// TwinCAT 3 PLC project IDPLC
// ProgramVersion: 3.1.4024.12
// libraries:
//   Recipe Management, * (System)
//   Tc2_Drive, * (Beckhoff Automation GmbH)
//   Tc2_EtherCAT, * (Beckhoff Automation GmbH)
//   Tc2_Math, * (Beckhoff Automation GmbH)
//   Tc2_MC2, * (Beckhoff Automation GmbH)
//   Tc2_NC, * (Beckhoff Automation GmbH)
//   Tc2_NcDrive, * (Beckhoff Automation GmbH)
//   Tc2_SerialCom, * (Beckhoff Automation GmbH)
//   Tc2_Standard, * (Beckhoff Automation GmbH)
//   Tc2_System, * (Beckhoff Automation GmbH)
//   Tc2_Utilities, * (Beckhoff Automation GmbH)
//   Tc3_Module, * (Beckhoff Automation GmbH)
// project tree:
//   DUTs/ DUT.TcDUT (not stored), DUT_SENSOR_DATAS_1.TcDUT (not stored), DUT_SENSOR_DATAS_8.TcDUT (not stored), DUT_SENSOR_DATAS_2.TcDUT (not stored), DUT_SENSOR_DATAS_3.TcDUT (not stored), DUT_SENSOR_DATAS_4.TcDUT (not stored), DUT_SENSOR_DATAS_5.TcDUT (not stored), DUT_SENSOR_DATAS_6.TcDUT (not stored), DUT_SENSOR_DATAS_7.TcDUT (not stored), Struct_M_Compensation.TcDUT, Struct_M_lakeshore.TcDUT (not stored), ST_P180.TcDUT (not stored), ST_P182.TcDUT (not stored), ST_P183.TcDUT (not stored)
//   GVLs/ Global_Variables.TcGVL, Variable_Configuration.TcGVL (not stored)
//   / PlcTask.TcTTO (not stored), RecipeManager.TcRMO (not stored)
//   POUs/0.UserMode/ F_GetSysTime.TcPOU (not stored), UserMode.TcPOU
//   POUs/1.CarrierMode/SingleCarrierMode/ SingleCarrierMode.TcPOU
//   POUs/2.SingleMotorMode/DebugMode/ DebugMode.TcPOU
//   POUs/CommonFB/ExternFB/ FB_LedShow.TcPOU (not stored), FB_PlcEmergencyStop.TcPOU (not stored)
//   POUs/CommonFB/MainFB/ FB_Move.TcPOU, FB_Power.TcPOU, FB_SetAxisPosition.TcPOU, FB_SetMotorAxisPosition.TcPOU, FB_Stop.TcPOU
//   POUs/ MAIN.TcPOU
//   POUs/RS232/ BackgroundEL.TcPOU (not stored), FB_SerialCom.TcPOU (not stored)

// ---- DUTs/Struct_M_Compensation.TcDUT
TYPE Struct_M_Compensation :
STRUCT
	Encoder:LREAL;
	LeftTop:LREAL;
	RightTop:LREAL;
	LeftBottom:LREAL;
	RightBottom:LREAL;
	LeftIn:LREAL;
	RightIn:LREAL;
	LeftOut:LREAL;
	RightOut:LREAL;
	InRange:BOOL;
END_STRUCT
END_TYPE

// ---- GVLs/Global_Variables.TcGVL
//{attribute 'Tc2GvlVarNames'}
VAR_GLOBAL
(*IDControl Ready*)
	IDControlReady:BOOL;
(*RecipeDescription*)
	RecipeSavedDate:STRING;
	RecipeDescription:STRING;
(*key Command*)
	btn_Power:BOOL;
	btn_PowerOn: BOOL;
	btn_PowerOff: BOOL;
(*Reset*)
	btn_Reset:BOOL;
(*Error Massage*)
	Error:BOOL;
	ErrorID:DINT;
	ErrorDescription:STRING;
(*加载配方参数*)
	LoadRecipeParameters:BOOL;
	loadParametersDone:BOOL;
(*Max Velocity Global*)
	MaxVelocityGlobalVelocity : LREAL;
(*设置光栅bias done *)	
	PositionBiasDone:BOOL;
(*回程差*)
	HysteresisError:LREAL;
(*Drive Status*)
	DriveStatus:DINT;//1:Drive Ready;2:Axis is in operation;0:Others
(*光栅漂移误差阈值*)
	LEDriftErrorThreshold:LREAL:=0.001;
(*Lag Distance threshold*)
	PosDiff_LeftTopLin: LREAL:=0.5;
	PosDiff_RightTopLin:LREAL:=0.5;
	PosDiff_LeftBottomLin:LREAL:=0.5;
	PosDiff_RightBottomLin:LREAL:=0.5;	
	PosDiff_LeftInLin: LREAL:=0.5;
	PosDiff_RightInLin:LREAL:=0.5;
	PosDiff_LeftOutLin:LREAL:=0.5;
	PosDiff_RightOutLin:LREAL:=0.5;
(*UserMode Threshold*)
	Threshold_UserTopPos: LREAL:=0.5;
	Threshold_UserBottomPos: LREAL:=0.5;
	Threshold_UserTBLeftPos: LREAL:=0.5;//TB=Top&Bottom
	Threshold_UserTBRightPos: LREAL:=0.5;
	Threshold_UserTopVelo: LREAL:=0.5;
	Threshold_UserBottomVelo: LREAL:=0.5;
	Threshold_UserTBLeftVelo: LREAL:=0.5;
	Threshold_UserTBRightVelo: LREAL:=0.5;
	Threshold_UserInPos: LREAL:=0.5;
	Threshold_UserOutPos: LREAL:=0.5;
	Threshold_UserIOLeftPos: LREAL:=0.5;//IO=In&Out
	Threshold_UserIORightPos: LREAL:=0.5;
	Threshold_UserInVelo: LREAL:=0.5;
	Threshold_UserOutVelo: LREAL:=0.5;
	Threshold_UserIOLeftVelo: LREAL:=0.5;
	Threshold_UserIORightVelo: LREAL:=0.5;
	//
	Range_UserTBTaperPos:LREAL:=4.01;
	Range_UserTBTaperVelo:LREAL:=1.01;
	Range_UserIOTaperPos:LREAL:=4.01;
	Range_UserIOTaperVelo:LREAL:=1.01;
(*UserMode*)
	//UserGapPositionNew:LREAL:=20;//target
	//UserGapVelocityNew:LREAL:=1;//target
(*DebugMode Threshold*)
	Threshold_TopPos_Debug: LREAL:=4;
	Threshold_BottomPos_Debug: LREAL:=4;
	Threshold_TBLeftPos_Debug: LREAL:=4;
	Threshold_TBRightPos_Debug: LREAL:=4;
	Threshold_InPos_Debug: LREAL:=4;
	Threshold_OutPos_Debug: LREAL:=4;
	Threshold_IOLeftPos_Debug: LREAL:=4;
	Threshold_IORightPos_Debug: LREAL:=4;
(*SingleCarrierMode threshold*)
	Threshold_TopPos_SingleCarrier: LREAL:=2;
	Threshold_BottomPos_SingleCarrier: LREAL:=2;
	Threshold_TBLeftPos_SingleCarrier: LREAL:=2;
	Threshold_TBRightPos_SingleCarrier: LREAL:=2;
	Threshold_TopVelo_SingleCarrier: LREAL:=2;
	Threshold_BottomVelo_SingleCarrier: LREAL:=2;
	Threshold_TBLeftVelo_SingleCarrier: LREAL:=2;
	Threshold_TBRightVelo_SingleCarrier: LREAL:=2;
	Threshold_InPos_SingleCarrier: LREAL:=2;
	Threshold_OutPos_SingleCarrier: LREAL:=2;
	Threshold_IOLeftPos_SingleCarrier: LREAL:=2;
	Threshold_IORightPos_SingleCarrier: LREAL:=2;
	Threshold_InVelo_SingleCarrier: LREAL:=2;
	Threshold_OutVelo_SingleCarrier: LREAL:=2;
	Threshold_IOLeftVelo_SingleCarrier: LREAL:=2;
	Threshold_IORightVelo_SingleCarrier: LREAL:=2;
	
	moveDoneLeftTop: BOOL;
	moveDoneRightTop: BOOL;
	moveDoneLeftBottom: BOOL;
	moveDoneRightBottom: BOOL;
	moveDoneLeftIn: BOOL;
	moveDoneRightIn: BOOL;
	moveDoneLeftOut: BOOL;
	moveDoneRightOut: BOOL;
	moveDoneAllAxis: BOOL;
	moveStatusLeftTop: BOOL;
	moveStatusRightTop: BOOL;
	moveStatusLeftBottom: BOOL;
	moveStatusRightBottom: BOOL;
	moveStatusLeftIn: BOOL;
	moveStatusRightIn: BOOL;
	moveStatusLeftOut: BOOL;
	moveStatusRightOut: BOOL;
	moveStatusAllAxis: BOOL;
	moveStatusAnyAxis: BOOL;
	
	moveDoneLeftTopMotor: BOOL;
	moveDoneRightTopMotor: BOOL;
	moveDoneLeftBottomMotor: BOOL;
	moveDoneRightBottomMotor: BOOL;
	moveDoneLeftInMotor: BOOL;
	moveDoneRightInMotor: BOOL;
	moveDoneLeftOutMotor: BOOL;
	moveDoneRightOutMotor: BOOL;
	moveDoneAllAxisMotor: BOOL;
	moveStatusLeftTopMotor: BOOL;
	moveStatusRightTopMotor: BOOL;
	moveStatusLeftBottomMotor: BOOL;
	moveStatusRightBottomMotor: BOOL;
	moveStatusLeftInMotor: BOOL;
	moveStatusRightInMotor: BOOL;
	moveStatusLeftOutMotor: BOOL;
	moveStatusRightOutMotor: BOOL;
	moveStatusAllAxisMotor: BOOL;
	moveStatusAnyAxisMotor: BOOL;
	(*input protection*)
	//
	min_UserGapPositionNew:LREAL:=10;
	max_UserGapPositionNew:LREAL:=200;
	inRange_UserGapPositionNew:BOOL;
	//LE protection position
	min_UserLEProtectionGapPosition:LREAL;
	min_ThresholdGapSoft2LEProtection:LREAL;
	max_UserLEProtectionGapPosition:LREAL;
	max_ThresholdGapSoft2LEProtection:LREAL;
	//
	min_UserGapVelocityNew:LREAL:=0;
	max_UserGapVelocityNew:LREAL:=2;
	inRange_UserGapVelocityNew:BOOL;
	//
	min_UserTaperPositionNew: LREAL:=0;;
	max_UserTaperPositionNew: LREAL:=1;
	inRange_UserTaperPositionNew: BOOL;
	//
	min_UserTaperVelocityNew: LREAL:=0;
	max_UserTaperVelocityNew: LREAL:=1;
	inRange_UserTaperVelocityNew: BOOL;
	
(*Compensation Value*)
	M_Compensation:ARRAY[1..18] OF Struct_M_Compensation
:=[
(Encoder:=0,		LeftTop:=0,			RightTop:=0,		LeftBottom:=0,			RightBottom:=0,			
					LeftIn:=0,			RightIn:=0,			LeftOut:=0,				RightOut:=0,			InRange:=FALSE),
(Encoder:=5,		LeftTop:=5,			RightTop:=5,		LeftBottom:=5,			RightBottom:=5,			
					LeftIn:=5,			RightIn:=5,			LeftOut:=5,				RightOut:=5,			InRange:=FALSE),
(Encoder:=6,		LeftTop:=6,			RightTop:=6,		LeftBottom:=6,			RightBottom:=6,			
					LeftIn:=6,			RightIn:=6,			LeftOut:=6,				RightOut:=6,			InRange:=FALSE),
(Encoder:=7,		LeftTop:=7,			RightTop:=7,		LeftBottom:=7,			RightBottom:=7,			
					LeftIn:=7,			RightIn:=7,			LeftOut:=7,				RightOut:=7,			InRange:=FALSE),
(Encoder:=8,		LeftTop:=8,			RightTop:=8,		LeftBottom:=8,			RightBottom:=8,			
					LeftIn:=8,			RightIn:=8,			LeftOut:=8,				RightOut:=8,			InRange:=FALSE),
(Encoder:=9,		LeftTop:=9,			RightTop:=9,		LeftBottom:=9,			RightBottom:=9,			
					LeftIn:=9,			RightIn:=9,			LeftOut:=9,				RightOut:=9,			InRange:=FALSE),
(Encoder:=10,		LeftTop:=10,		RightTop:=10,		LeftBottom:=10,			RightBottom:=10,			
					LeftIn:=10,			RightIn:=10,		LeftOut:=10,			RightOut:=10,			InRange:=FALSE),
(Encoder:=11,		LeftTop:=11,		RightTop:=11,		LeftBottom:=11,			RightBottom:=11,			
					LeftIn:=11,			RightIn:=11,		LeftOut:=11,			RightOut:=11,			InRange:=FALSE),
(Encoder:=12,		LeftTop:=12,		RightTop:=12,		LeftBottom:=12,			RightBottom:=12,			
					LeftIn:=12,			RightIn:=12,		LeftOut:=12,			RightOut:=12,			InRange:=FALSE),
(Encoder:=13,		LeftTop:=13,		RightTop:=13,		LeftBottom:=13,			RightBottom:=13,			
					LeftIn:=13,			RightIn:=13,		LeftOut:=13,			RightOut:=13,			InRange:=FALSE),
(Encoder:=15,		LeftTop:=15,		RightTop:=15,		LeftBottom:=15,			RightBottom:=15,			
					LeftIn:=15,			RightIn:=15,		LeftOut:=15,			RightOut:=15,			InRange:=FALSE),
(Encoder:=20,		LeftTop:=20,		RightTop:=20,		LeftBottom:=20,			RightBottom:=20,			
					LeftIn:=20,			RightIn:=20,		LeftOut:=20,			RightOut:=20,			InRange:=FALSE),
(Encoder:=22,		LeftTop:=22,		RightTop:=22,		LeftBottom:=22,			RightBottom:=22,			
					LeftIn:=22,			RightIn:=22,		LeftOut:=22,			RightOut:=22,			InRange:=FALSE),
(Encoder:=30,		LeftTop:=30,		RightTop:=30,		LeftBottom:=30,			RightBottom:=30,			
					LeftIn:=30,			RightIn:=30,		LeftOut:=30,			RightOut:=30,			InRange:=FALSE),
(Encoder:=40,		LeftTop:=40,		RightTop:=40,		LeftBottom:=40,			RightBottom:=40,			
					LeftIn:=40,			RightIn:=40,		LeftOut:=40,			RightOut:=40,			InRange:=FALSE),
(Encoder:=50,		LeftTop:=50,		RightTop:=50,		LeftBottom:=50,			RightBottom:=50,			
					LeftIn:=50,			RightIn:=50,		LeftOut:=50,			RightOut:=50,			InRange:=FALSE),
(Encoder:=100,		LeftTop:=100,		RightTop:=100,		LeftBottom:=100,		RightBottom:=100,			
					LeftIn:=100,		RightIn:=100,		LeftOut:=100,			RightOut:=100,			InRange:=FALSE),
(Encoder:=3000.001,	LeftTop:=3000.001,	RightTop:=3000.001,	LeftBottom:=3000.001,	RightBottom:=3000.001,			
					LeftIn:=3000.001,	RightIn:=3000.001,	LeftOut:=3000.001,		RightOut:=3000.001,			InRange:=FALSE)];
(*simulation OR NOT*)
	simulation:BOOL;
(*USELinearEncoeder*)
	USELinearEncoder:BOOL:=TRUE;
(*restartTwinCAT*)
	m_restartTC:BOOL;
(*Plc_EmergencyStop *)
	Plc_EmergencyStop  AT %Q*:BOOL:=TRUE;
(*硬急停*)
	Hardware_EmergencyStop :BOOL:=TRUE;
(*LED*)
	Led_Run  AT %Q*:BOOL;
	Led_Error  AT %Q*:BOOL;
(*LimitSwitch*)
	LS_LeftTop_Far  :BOOL;
	LS_LeftTop_Near  :BOOL;
	LS_RightTop_Far  :BOOL;
	LS_RightTop_Near  :BOOL;
	LS_LeftBottom_Far  :BOOL;
	LS_LeftBottom_Near  :BOOL;
	LS_RightBottom_Far :BOOL;
	LS_RightBottom_Near  :BOOL;
	Unreach_LS_Far:BOOL;
	Unreach_LS_Near:BOOL;
	LS_LeftIn_Far  :BOOL;
	LS_LeftIn_Near  :BOOL;
	LS_RightIn_Far  :BOOL;
	LS_RightIn_Near  :BOOL;
	LS_LeftOut_Far  :BOOL;
	LS_LeftOut_Near  :BOOL;
	LS_RightOut_Far :BOOL;
	LS_RightOut_Near  :BOOL;
(*kill switch*)
	KS_LeftTop_Far_Contact1:BOOL;
	KS_LeftTop_Far_Contact2:BOOL;
	KS_RightTop_Far_Contact1:BOOL;
	KS_RightTop_Far_Contact2:BOOL;
	KS_LeftBottom_Far_Contact1:BOOL;
	KS_LeftBottom_Far_Contact2:BOOL;
	KS_RightBottom_Far_Contact1:BOOL;
	KS_RightBottom_Far_Contact2:BOOL;
	
	KS_LeftTop_Near_Contact1:BOOL;
	KS_LeftTop_Near_Contact2:BOOL;
	KS_RightTop_Near_Contact1:BOOL;
	KS_RightTop_Near_Contact2:BOOL;
	KS_LeftBottom_Near_Contact1:BOOL;
	KS_LeftBottom_Near_Contact2:BOOL;
	KS_RightBottom_Near_Contact1:BOOL;
	KS_RightBottom_Near_Contact2:BOOL;
	
	KS_LeftIn_Far_Contact1:BOOL;
	KS_LeftIn_Far_Contact2:BOOL;
	KS_RightIn_Far_Contact1:BOOL;
	KS_RightIn_Far_Contact2:BOOL;
	KS_LeftOut_Far_Contact1:BOOL;
	KS_LeftOut_Far_Contact2:BOOL;
	KS_RightOut_Far_Contact1:BOOL;
	KS_RightOut_Far_Contact2:BOOL;
	
	KS_LeftIn_Near_Contact1:BOOL;
	KS_LeftIn_Near_Contact2:BOOL;
	KS_RightIn_Near_Contact1:BOOL;
	KS_RightIn_Near_Contact2:BOOL;
	KS_LeftOut_Near_Contact1:BOOL;
	KS_LeftOut_Near_Contact2:BOOL;
	KS_RightOut_Near_Contact1:BOOL;
	KS_RightOut_Near_Contact2:BOOL;
(*E-STOP*)
	KS_CabinetEmergency_contact1:BOOL;
	KS_CabinetEmergency_contact2:BOOL;
	KS_handEmergency1_Contact1:BOOL;
	KS_handEmergency1_Contact2:BOOL;
	KS_handEmergency2_Contact1:BOOL;
	KS_handEmergency2_Contact2:BOOL;
	KS_softEmergency2_Contact:BOOL;
(*aixs_ref*)
	LeftTopLin: axis_ref;
	RightTopLin:axis_ref;
	LeftBottomLin:axis_ref;
	RightBottomLin:axis_ref;
	LeftInLin: axis_ref;
	RightInLin:axis_ref;
	LeftOutLin:axis_ref;
	RightOutLin:axis_ref;
(*aixs_ref-motor*)
	LeftTopMotor: axis_ref;
	RightTopMotor:axis_ref;
	LeftBottomMotor:axis_ref;
	RightBottomMotor:axis_ref;
	LeftInMotor: axis_ref;
	RightInMotor:axis_ref;
	LeftOutMotor:axis_ref;
	RightOutMotor:axis_ref;
(*axis Position*)
	Pos_LeftTopLin: LREAL;
	Pos_RightTopLin:LREAL;
	Pos_LeftBottomLin:LREAL;
	Pos_RightBottomLin:LREAL;
	Pos_LeftInLin: LREAL;
	Pos_RightInLin:LREAL;
	Pos_LeftOutLin:LREAL;
	Pos_RightOutLin:LREAL;
(*axis Position-motor*)
	Pos_LeftTopMotor: LREAL;
	Pos_RightTopMotor:LREAL;
	Pos_LeftBottomMotor:LREAL;
	Pos_RightBottomMotor:LREAL;
	Pos_LeftInMotor: LREAL;
	Pos_RightInMotor:LREAL;
	Pos_LeftOutMotor:LREAL;
	Pos_RightOutMotor:LREAL;
(*axis Position-Delta*)
	DeltaPos_LeftTop: LREAL;
	DeltaPos_RightTop:LREAL;
	DeltaPos_LeftBottom:LREAL;
	DeltaPos_RightBottom:LREAL;
	DeltaPos_LeftIn: LREAL;
	DeltaPos_RightIn:LREAL;
	DeltaPos_LeftOut:LREAL;
	DeltaPos_RightOut:LREAL;
(*axis Position-Threshold*)
	ThresholdDeltaPos_LeftTop: LREAL:=0.2;
	ThresholdDeltaPos_RightTop:LREAL:=0.2;
	ThresholdDeltaPos_LeftBottom:LREAL:=0.2;
	ThresholdDeltaPos_RightBottom:LREAL:=0.2;
	ThresholdDeltaPos_LeftIn: LREAL:=0.2;
	ThresholdDeltaPos_RightIn:LREAL:=0.2;
	ThresholdDeltaPos_LeftOut:LREAL:=0.2;
	ThresholdDeltaPos_RightOut:LREAL:=0.2;
(*axis Velocity*)
	Velo_LeftTopLin: LREAL;
	Velo_RightTopLin:LREAL;
	Velo_LeftBottomLin:LREAL;
	Velo_RightBottomLin:LREAL;
	Velo_LeftInLin: LREAL;
	Velo_RightInLin:LREAL;
	Velo_LeftOutLin:LREAL;
	Velo_RightOutLin:LREAL;
(*axis Velocity-motor*)
	Velo_LeftTopMotor: LREAL;
	Velo_RightTopMotor:LREAL;
	Velo_LeftBottomMotor:LREAL;
	Velo_RightBottomMotor:LREAL;
	Velo_LeftInMotor: LREAL;
	Velo_RightInMotor:LREAL;
	Velo_LeftOutMotor:LREAL;
	Velo_RightOutMotor:LREAL;
(*axis Velocity-Delta*)
	DeltaVelo_LeftTop: LREAL;
	DeltaVelo_RightTop:LREAL;
	DeltaVelo_LeftBottom:LREAL;
	DeltaVelo_RightBottom:LREAL;
	DeltaVelo_LeftIn: LREAL;
	DeltaVelo_RightIn:LREAL;
	DeltaVelo_LeftOut:LREAL;
	DeltaVelo_RightOut:LREAL;
(*axis Velocity-ThresholdDelta*)
	ThresholdDeltaVelo_LeftTop: LREAL:=0.1;
	ThresholdDeltaVelo_RightTop:LREAL:=0.1;
	ThresholdDeltaVelo_LeftBottom:LREAL:=0.1;
	ThresholdDeltaVelo_RightBottom:LREAL:=0.1;
	ThresholdDeltaVelo_LeftIn: LREAL:=0.1;
	ThresholdDeltaVelo_RightIn:LREAL:=0.1;
	ThresholdDeltaVelo_LeftOut:LREAL:=0.1;
	ThresholdDeltaVelo_RightOut:LREAL:=0.1;
(*axis Torque-motor*)
	Torque_LeftTopLin: LREAL;
	Torque_RightTopLin:LREAL;
	Torque_LeftBottomLin:LREAL;
	Torque_RightBottomLin:LREAL;
	Torque_LeftInLin: LREAL;
	Torque_RightInLin:LREAL;
	Torque_LeftOutLin:LREAL;
	Torque_RightOutLin:LREAL;
(*axis Torque-motor*)
	Torque_LeftTopMotor: LREAL;
	Torque_RightTopMotor:LREAL;
	Torque_LeftBottomMotor:LREAL;
	Torque_RightBottomMotor:LREAL;
	Torque_LeftInMotor: LREAL;
	Torque_RightInMotor:LREAL;
	Torque_LeftOutMotor:LREAL;
	Torque_RightOutMotor:LREAL;
(*axis Torque-Delta*)
	DeltaTorque_LeftTop: LREAL;
	DeltaTorque_RightTop:LREAL;
	DeltaTorque_LeftBottom:LREAL;
	DeltaTorque_RightBottom:LREAL;
	DeltaTorque_LeftIn: LREAL;
	DeltaTorque_RightIn:LREAL;
	DeltaTorque_LeftOut:LREAL;
	DeltaTorque_RightOut:LREAL;
(*Lag Distance*)
	PosDiff_LeftTopLin_actual: LREAL;
	PosDiff_RightTopLin_actual:LREAL;
	PosDiff_LeftBottomLin_actual:LREAL;
	PosDiff_RightBottomLin_actual:LREAL;
	PosDiff_LeftInLin_actual: LREAL;
	PosDiff_RightInLin_actual:LREAL;
	PosDiff_LeftOutLin_actual:LREAL;
	PosDiff_RightOutLin_actual:LREAL;
(*Lag Distance-Motor*)
	PosDiff_LeftTopMotor_actual: LREAL;
	PosDiff_RightTopMotor_actual:LREAL;
	PosDiff_LeftBottomMotor_actual:LREAL;
	PosDiff_RightBottomMotor_actual:LREAL;
	PosDiff_LeftInMotor_actual: LREAL;
	PosDiff_RightInMotor_actual:LREAL;
	PosDiff_LeftOutMotor_actual:LREAL;
	PosDiff_RightOutMotor_actual:LREAL;
(*Delta LagDistance*)
	DeltaPosDiff_LeftTop_actual: LREAL;
	DeltaPosDiff_RightTop_actual:LREAL;
	DeltaPosDiff_LeftBottom_actual:LREAL;
	DeltaPosDiff_RightBottom_actual:LREAL;
	DeltaPosDiff_LeftIn_actual: LREAL;
	DeltaPosDiff_RightIn_actual:LREAL;
	DeltaPosDiff_LeftOut_actual:LREAL;
	DeltaPosDiff_RightOut_actual:LREAL;
(*****************singleCarrier Mode*******************************)
(**)
	TopPositionActual:LREAL;
	TopVelocityActual:LREAL;
	BottomPositionActual:LREAL;
	BottomVelocityActual:LREAL;
	TopMoveIndicator:DINT:=0;
	(*1=OPEN;0=NOTMOVE;-1=CLOSE*)
	BottomMoveIndicator:DINT:=0;
	(*1=OPEN;0=NOTMOVE;-1=CLOSE*)
	InPositionActual:LREAL;
	InVelocityActual:LREAL;
	OutPositionActual:LREAL;
	OutVelocityActual:LREAL;
	InMoveIndicator:DINT:=0;
	(*1=OPEN;0=NOTMOVE;-1=CLOSE*)
	OutMoveIndicator:DINT:=0;
	(*1=OPEN;0=NOTMOVE;-1=CLOSE*)

(******************SingleCarrier***********************************)
	Diff_TopPos_actual: LREAL;
	Diff_BottomPos_actual: LREAL;
	Diff_TBLeftPos_actual: LREAL;
	Diff_TBRightPos_actual: LREAL;
	Diff_TopVelo_actual:  LREAL;
	Diff_BottomVelo_actual: LREAL;
	Diff_TBLeftVelo_actual: LREAL;
	Diff_TBRightVelo_actual:  LREAL;
	Diff_InPos_actual: LREAL;
	Diff_OutPos_actual: LREAL;
	Diff_IOLeftPos_actual: LREAL;
	Diff_IORightPos_actual: LREAL;
	Diff_InVelo_actual:  LREAL;
	Diff_OutVelo_actual: LREAL;
	Diff_IOLeftVelo_actual: LREAL;
	Diff_IORightVelo_actual:  LREAL;

(******************UserMode*********************)
	Diff_UserTopPos_actual: LREAL;
	Diff_UserBottomPos_actual: LREAL;
	Diff_UserTBLeftPos_actual: LREAL;
	Diff_UserTBRightPos_actual: LREAL;
	Diff_UserTopVelo_actual:  LREAL;
	Diff_UserBottomVelo_actual: LREAL;
	Diff_UserTBLeftVelo_actual: LREAL;
	Diff_UserTBRightVelo_actual:  LREAL;
	Diff_UserInPos_actual: LREAL;
	Diff_UserOutPos_actual: LREAL;
	Diff_UserIOLeftPos_actual: LREAL;
	Diff_UserIORightPos_actual: LREAL;
	Diff_UserInVelo_actual:  LREAL;
	Diff_UserOutVelo_actual: LREAL;
	Diff_UserIOLeftVelo_actual: LREAL;
	Diff_UserIORightVelo_actual:  LREAL;
(******************************************)
	TaperFunctionSolidOn:BOOL;//该ID是否有taper需求，taper总开关，只在参数表生效
	TaperOrNot:BOOL;
	UserTaperPositionActual:LREAL;
	UserTaperVelocityActual:LREAL;
	UserTBTaperPositionActual:LREAL;
	UserTBTaperVelocityActual:LREAL;
	UserIOTaperPositionActual:LREAL;
	UserIOTaperVelocityActual:LREAL;
(***********************Power status and couple statatus***********************)
	st_Power:BOOL;
	st_Couple:DINT;
(************************FB***********************)
	FB_Power:FB_Power;
	FB_PlcEmergencyStop: FB_PlcEmergencyStop;
	FB_Move:FB_Move;
	FB_Stop:FB_Stop;
	(*SingleCarrierMode All Move/Stop*)
	FB_Move_Top:FB_Move;
	FB_Stop_Top:FB_Stop;
	FB_Move_Bottom:FB_Move;
	FB_Stop_Bottom:FB_Stop;
	FB_Move_In:FB_Move;
	FB_Stop_In:FB_Stop;
	FB_Move_Out:FB_Move;
	FB_Stop_Out:FB_Stop;

	M_CompensationNumber:INT;
	M_DisplayNumber:INT;
		
	(*Conpensation Position Target*)
	LeftTopLinPositionNew:LREAL;
	LeftBottomLinPositionNew:LREAL;
	RightTopLinPositionNew:LREAL;
	RightBottomLinPositionNew:LREAL;
	LeftInLinPositionNew:LREAL;
	LeftOutLinPositionNew:LREAL;
	RightInLinPositionNew:LREAL;
	RightOutLinPositionNew:LREAL;
	(*考虑到回程差后，运动到临时位置*)
	LeftTopLinPositionNew_temporary :LREAL;
	LeftBottomLinPositionNew_temporary:LREAL;
	RightTopLinPositionNew_temporary:LREAL;
	RightBottomLinPositionNew_temporary:LREAL;
	LeftInLinPositionNew_temporary :LREAL;
	LeftOutLinPositionNew_temporary:LREAL;
	RightInLinPositionNew_temporary:LREAL;
	RightOutLinPositionNew_temporary:LREAL;
	(*Display Position*)
	LeftTopLinPositionDisplay:LREAL;
	LeftBottomLinPositionDisplay:LREAL;
	RightTopLinPositionDisplay:LREAL;
	RightBottomLinPositionDisplay:LREAL;
	LeftInLinPositionDisplay:LREAL;
	LeftOutLinPositionDisplay:LREAL;
	RightInLinPositionDisplay:LREAL;
	RightOutLinPositionDisplay:LREAL;
	(*Display Velocity*)
	LeftTopLinVelocityDisplay:LREAL;
	LeftBottomLinVelocityDisplay:LREAL;
	RightTopLinVelocityDisplay:LREAL;
	RightBottomLinVelocityDisplay:LREAL;
	LeftInLinVelocityDisplay:LREAL;
	LeftOutLinVelocityDisplay:LREAL;
	RightInLinVelocityDisplay:LREAL;
	RightOutLinVelocityDisplay:LREAL;
	(*temperature sensors*)
	thermocouple AT %I*:ARRAY[1..12]OF  DINT;
	shieldPt100  AT %I*:ARRAY[1..12]OF INT;
	thermocouple_Celsius:ARRAY[1..12]OF  LREAL;
	shieldPt100_Celsius  :ARRAY[1..12]OF LREAL;
	huoer_Celsius AT %I* :ARRAY[1..3]OF INT;
	(**)
	lakeshorePt100  AT %I*:ARRAY[1..12]OF INT;(*16*×èÖµ*)
	lakeshorePt100_Resistance :ARRAY[1..12]OF LREAL;(*ÉãÊÏÎÂ¶È*)
	lakeshorePt100_Celsius  :ARRAY[1..12]OF LREAL;(*ÉãÊÏÎÂ¶È*)
	temperatureCompensationValue:LREAL:=6;
	testSensors  AT %I*:ARRAY[1..4]OF INT;

(******RS232************)
	RxBufferEL			: ComBuffer;	(* Receive data buffer; used with all receive function blocks *)
	TxBufferEL			: ComBuffer;	(* Transmit data buffer; used with all receive function blocks *)

END_VAR

// ---- POUs/0.UserMode/UserMode.TcPOU
PROGRAM UserMode
VAR_INPUT
	UserGapPositionNew:LREAL:=20;//target
	UserGapVelocityNew:LREAL:=1;//target
		(**)
	btn_UserGapMove:BOOL;
	btn_UserGapStop:BOOL;
END_VAR
VAR	
	USE_SingleAxis_Compensation:BOOL:=TRUE;
(*GapMode*)

	UserGapPositionDisplay:LREAL;//current
	UserGapVelocityDisplay:LREAL;//current
	UserTaperPositionNew:LREAL:=0;//target
	UserTaperVelocityNew:LREAL:=0.1;//target
	UserTaperPositionDisplay:LREAL;//current
	UserTaperVelocityDisplay:LREAL;//target
	UserGapPositionDisplay_FromLeftTop:LREAL;
	UserGapPositionDisplay_FromLeftBottom:LREAL;
	UserGapPositionDisplay_FromLeftIn:LREAL;
	UserGapPositionDisplay_FromLeftOut:LREAL;
	//
	UserRightGapPositionNew:LREAL;
	UserRightGapVelocityNew:LREAL;
	UserRightGapPositionDisplay:LREAL;
	UserRightGapVelocityDisplay:LREAL;
	UserRightGapPositionDisplay_FromRightTop:LREAL;
	UserRightGapPositionDisplay_FromRightBottom:LREAL;
	UserRightGapPositionDisplay_FromRightIn:LREAL;
	UserRightGapPositionDisplay_FromRightOut:LREAL;

	(*Var*)
	fb_ton1:TON;
	fb_ton2:TON;
	fb_ton3:TON;
	fb_ton4:TON;
	fb_ton5:TON;
	fb_ton6:TON;
	(*Status*)
	State:DINT;
	Busy:BOOL;
	InitPowerDone:BOOL;
	InitCompensationDatasDone:BOOL;
	(*FB*)
	m_state: DINT;
	n_state: DINT;
	s_state: DINT;
	(*¼ì²âµ½ÏÞÎ»£¬»Ö¸´Move×´Ì¬*)
	FTrig_ReachLS: F_TRIG;
	FTrig_btn_GapMove: F_TRIG;
	GapOutRange: BOOL;
	(*PowerOff*)
	d_state: DINT;
	i: INT;
	j: INT;
	k: INT;
	moni_State:DINT;
	TargetPosLessThanCurrentPos:BOOL;
	TargetLTPosLessThanCurrentLTPos:BOOL;
	TargetRTPosLessThanCurrentRTPos:BOOL;
	TargetLBPosLessThanCurrentLBPos:BOOL;
	TargetRBPosLessThanCurrentRBPos:BOOL;
	TargetLIPosLessThanCurrentLIPos:BOOL;
	TargetRIPosLessThanCurrentRIPos:BOOL;
	TargetLOPosLessThanCurrentLOPos:BOOL;
	TargetROPosLessThanCurrentROPos:BOOL;
	PositiveMoving:BOOL;
	HysteresisMoving:BOOL;
	NoneHysteresisMoving:BOOL;
	(*Spectroscopy scanning Mode*)
	IsSSMotionMode:BOOL;
	RegularMotionMode:BOOL;
	SSMotionMode:BOOL;
	SS_StepSize:LREAL:=0.001;
	SS_StepNumber:INT:=10;
	SS_StepVelocity:LREAL:=1;
	SS_Move:BOOL;
	SS_Stop:BOOL;
	SS_MoveState:DINT;
	SS_StopState:DINT;
	SS_currentStep:DINT:=0;
	SS_StepSystemTime_Begin:ARRAY[0..100] OF ULINT;
	SS_StepSystemTime_End:ARRAY[0..100] OF ULINT;
	SS_StepCountTime:ARRAY[0..100] OF ULINT;
	SS_TimeCountBegin:BOOL;
	m: INT;
	SS_TON: TON;
	StepEachTime:TIME;
	StepEachTime_ms:INT:=1000;//ms
	SS_OTSTRUCT :OTSTRUCT ;
	SS_StartPositionDisplay:LREAL;
	RTRG_SS_StartPositionDisplay:R_TRIG;
	SS_InitStartPositionDone:BOOL;
	//
	min_SS_StepSize	: LREAL:=0;
	max_SS_StepSize	: LREAL:=200;
	inRange_SS_StepSize	: BOOL;
	//
	min_SS_StepNumber	: INT:=1;
	max_SS_StepNumber	: INT:=1000;
	inRange_SS_StepNumber	: BOOL;
	//
	min_SS_StepVelocity:LREAL:=0;
	max_SS_StepVelocity:LREAL:=1;
	inRange_SS_StepVelocity:BOOL;
	//
	min_StepEachTime_ms:INT:=100;
	max_StepEachTime_ms:INT:=10000;
	inRange_StepEachTime_ms:BOOL;
	l: INT;
	Threshold_UserTopPos_PLC: LREAL;
	Threshold_UserTopVelo_PLC: LREAL;
	Threshold_UserBottomPos_PLC: LREAL;
	Threshold_UserBottomVelo_PLC: LREAL;
	Threshold_UserTBLeftPos_PLC: LREAL;
	Threshold_UserTBLeftVelo_PLC: LREAL;
	Threshold_UserTBRightPos_PLC: LREAL;
	Threshold_UserTBRightVelo_PLC: LREAL;
	Threshold_UserInPos_PLC: LREAL;
	Threshold_UserInVelo_PLC: LREAL;
	Threshold_UserOutPos_PLC: LREAL;
	Threshold_UserOutVelo_PLC: LREAL;
	Threshold_UserIOLeftPos_PLC: LREAL;
	Threshold_UserIOLeftVelo_PLC: LREAL;
	Threshold_UserIORightPos_PLC: LREAL;
	Threshold_UserIORightVelo_PLC: LREAL;
	testa: BOOL;
	testb: BOOL;
	Threshold_GapChangeFlag: LREAL:=0.001;
	Threshold_TaperChangeFlag: LREAL:=0.005;
	TaperAndGapSafetyfactor: LREAL:=1;
	TaperAndGapSafetyScale:LREAL:=0.42;//IAU=0.41,IVU=0.32,CPMU=0.33,IAMW=0.42
	TaperAndGapSafetyMinGapMargin:LREAL:=0.4;

		//Global Chain protection-MPS
	Global_ChainProtection_MPS_StorageRingReady:BOOL;
	Global_ChainProtection_MPS_On: BOOL;
	Global_ChainProtection_MPS_MaxGapValue: LREAL;
	Global_ChainProtection_MPS_MoveVelocity: LREAL;
	Global_ChainProtection_MPS_Done: BOOL;
	//Global_ChainProtection_Error: BOOL;
	//Global_ChainProtection_ErrorID: INT;
	//Global_ChainProtection_ErrorDescription: STRING;
	Global_ChainProtection_MPS_ManualOperation:BOOL:=TRUE;
	Global_ChainProtection_MPS_FTRIG:F_TRIG;
	Global_ChainProtection_MPS_FTRIG_Manul:F_TRIG;
	Global_ChainProtection_MPS_TON:TON;
	Global_ChainProtection_MPS_Triggered:BOOL;
	Global_ChainProtection_MPS_In:BOOL;
	Global_ChainProtection_MPS_In1 AT%I* :BOOL;//下降沿表示触发,EL1008
	Global_ChainProtection_MPS_In2 AT%I* :BOOL;
	Global_ChainProtection_MPS_State:DINT;
	Global_ChainProtection_MPS_Out1 AT%Q* :BOOL;//上升沿标识到达最大间隙，连锁保护成功,EL2624
	Global_ChainProtection_MPS_Out2 AT%Q* :BOOL;
	Global_ChainProtection_MPS_TON_Stop2Move:TON;
	Global_ChainProtection_MPS_TON_Stop2Move_InTaperMode:TON;
	Global_ChainProtection_MPS_TON_Power2Move:TON;
	//Global Chain protection-EPS
	Global_ChainProtection_EPS_BeamLineReady:BOOL;
	Global_ChainProtection_EPS_On: BOOL;
	Global_ChainProtection_EPS_MaxGapValue: LREAL;
	Global_ChainProtection_EPS_MoveVelocity: LREAL;
	Global_ChainProtection_EPS_Done: BOOL;
	//Global_ChainProtection_Error: BOOL;
	//Global_ChainProtection_ErrorID: INT;
	//Global_ChainProtection_ErrorDescription: STRING;
	Global_ChainProtection_EPS_ManualOperation:BOOL:=TRUE;
	Global_ChainProtection_EPS_FTRIG:F_TRIG;
	Global_ChainProtection_EPS_FTRIG_Manul:F_TRIG;
	Global_ChainProtection_EPS_TON:TON;
	Global_ChainProtection_EPS_Triggered:BOOL;
	Global_ChainProtection_EPS_In:BOOL;
	Global_ChainProtection_EPS_In1 AT%I* :BOOL;//下降沿表示触发,EL1124
	Global_ChainProtection_EPS_In2 AT%I* :BOOL;
	Global_ChainProtection_EPS_State:DINT;
	Global_ChainProtection_EPS_Out1 AT%Q* :BOOL;//上升沿标识到达最大间隙，连锁保护成功,EL2124
	Global_ChainProtection_EPS_Out2 AT%Q* :BOOL;
	Global_ChainProtection_EPS_TON_Stop2Move:TON;
	Global_ChainProtection_EPS_TON_Stop2Move_InTaperMode:TON;
	Global_ChainProtection_EPS_TON_Power2Move:TON;
	//
	Threshold_motorsTargetPosCalculate: LREAL;
	//
	LeftTopLinPositionNewTemp: LREAL;
	RightTopLinPositionNewTemp: LREAL;
	LeftBottomLinPositionNewTemp: LREAL;
	RightBottomLinPositionNewTemp: LREAL;
	LeftInLinPositionNewTemp: LREAL;
	RightInLinPositionNewTemp: LREAL;
	LeftOutLinPositionNewTemp: LREAL;
	RightOutLinPositionNewTemp: LREAL;
	//OneKeyToMaxGap
	btn_OneKeyToMaxGap:BOOL;
	OneKeyToMaxGap_RTRIG:R_TRIG;
	OneKeyToMaxGap_TON:TON;
	OneKeyToMaxGap_Triggered:BOOL;
	OneKeyToMaxGap_State:DINT;
	OneKeyToMaxGap_TON_Stop2Move:TON;
	OneKeyToMaxGap_TON_Stop2Move_InTaperMode:TON;
	OneKeyToMaxGap_TON_Power2Move:TON;
	OneKeyToMaxGap_Done:BOOL;
END_VAR

IF NOT PositionBiasDone THEN
	RETURN;
END_IF
IF NOT loadParametersDone THEN
	RETURN;
END_IF
(*btn_Power On/Off*)
IF btn_Power AND NOT st_Power THEN
	btn_PowerOn:=TRUE;
	btn_Power:=FALSE;
END_IF
IF btn_Power AND st_Power THEN
	btn_PowerOff:=TRUE;
	btn_Power:=FALSE;
END_IF
IF btn_PowerOn THEN
	A_PowerOn();
END_IF
IF btn_PowerOff THEN
	A_PowerOff();
END_IF

(*监控四轴位置速度等*)
A_MonitoringAllAxis();

(*补偿数据处理*)
A_InitCompensationData();

(*常规磁间隙开合*)
IF RegularMotionMode AND NOT SSMotionMode THEN
	A_RegularMotion();
END_IF

(*
(*Spectroscopy scanning Mode*)
IF IsSSMotionMode THEN
	SSMotionMode:=TRUE;
	RegularMotionMode:=FALSE;
ELSE
	SSMotionMode:=FALSE;
	RegularMotionMode:=TRUE;
END_IF
IF	SSMotionMode AND NOT RegularMotionMode THEN
	A_SpectroscopyScanningMotion();
END_IF
*)
(*A_CheckMotorsPos*)
A_CheckMotorsPos();

(*GlobalChainProtection*)
A_GlobalChainProtection_MPS();
A_GlobalChainProtection_EPS();
(*A_OneKeyToMaxGap*)
A_OneKeyToMaxGap();

ACTION A_CheckMotorsPos:
//
//目标位置速度超出阈值判断
//
//gap posiion
IF UserGapPositionNew<min_UserGapPositionNew OR UserGapPositionNew>max_UserGapPositionNew THEN
	inRange_UserGapPositionNew:=FALSE;
END_IF
IF UserGapPositionNew>=min_UserGapPositionNew AND UserGapPositionNew<=max_UserGapPositionNew THEN
	inRange_UserGapPositionNew:=TRUE;
END_IF
//gap velocity
IF UserGapVelocityNew<min_UserGapVelocityNew OR UserGapVelocityNew>max_UserGapVelocityNew THEN
	inRange_UserGapVelocityNew:=FALSE;
END_IF
IF UserGapVelocityNew>=min_UserGapVelocityNew AND UserGapVelocityNew<=max_UserGapVelocityNew THEN
	inRange_UserGapVelocityNew:=TRUE;
END_IF
//taper position
IF UserTaperPositionNew<min_UserTaperPositionNew OR UserTaperPositionNew>max_UserTaperPositionNew THEN
	inRange_UserTaperPositionNew:=FALSE;
END_IF
IF UserTaperPositionNew>=min_UserTaperPositionNew AND UserTaperPositionNew<=max_UserTaperPositionNew THEN
	inRange_UserTaperPositionNew:=TRUE;
END_IF
//taper velocity
IF UserTaperVelocityNew<min_UserTaperVelocityNew OR UserTaperVelocityNew>max_UserTaperVelocityNew THEN
	inRange_UserTaperVelocityNew:=FALSE;
END_IF
IF UserTaperVelocityNew>=min_UserTaperVelocityNew AND UserTaperVelocityNew<=max_UserTaperVelocityNew THEN
	inRange_UserTaperVelocityNew:=TRUE;
END_IF
//SS Mode
IF SS_StepSize<min_SS_StepSize OR SS_StepSize>max_SS_StepSize THEN
	inRange_SS_StepSize:=FALSE;
END_IF
IF SS_StepSize>=min_SS_StepSize AND SS_StepSize<=max_SS_StepSize THEN
	inRange_SS_StepSize:=TRUE;
END_IF
IF SS_StepNumber<min_SS_StepNumber OR SS_StepNumber>max_SS_StepNumber THEN
	inRange_SS_StepNumber:=FALSE;
END_IF
IF SS_StepNumber>=min_SS_StepNumber AND SS_StepNumber<=max_SS_StepNumber THEN
	inRange_SS_StepNumber:=TRUE;
END_IF
IF SS_StepVelocity<min_SS_StepVelocity OR SS_StepVelocity>max_SS_StepVelocity THEN
	inRange_SS_StepVelocity:=FALSE;
END_IF
IF SS_StepVelocity>=min_SS_StepVelocity AND SS_StepVelocity<=max_SS_StepVelocity THEN
	inRange_SS_StepVelocity:=TRUE;
END_IF
IF StepEachTime_ms<min_StepEachTime_ms OR StepEachTime_ms>max_StepEachTime_ms THEN
	inRange_StepEachTime_ms:=FALSE;
END_IF
IF StepEachTime_ms>=min_StepEachTime_ms AND StepEachTime_ms<=max_StepEachTime_ms THEN
	inRange_StepEachTime_ms:=TRUE;
END_IF


//
//输入速度和位置保护
//
IF btn_UserGapMove  AND NOT SSMotionMode AND RegularMotionMode THEN
	IF NOT inRange_UserGapPositionNew THEN
		btn_UserGapStop:=TRUE;
		btn_UserGapMove:=FALSE;
		Error:=TRUE;
		ErrorId:=801;
		ErrorDescription:='target Gap position out of range,please check';
		RETURN;
	ELSE
		//btn_UserGapStop:=FALSE;
		Error:=FALSE;
		ErrorId:=0;
		ErrorDescription:='';	
	END_IF
	IF NOT inRange_UserGapVelocityNew THEN
		btn_UserGapStop:=TRUE;
		btn_UserGapMove:=FALSE;
		Error:=TRUE;
		ErrorId:=802;
		ErrorDescription:='target Gap velocity out of range,please check';
		RETURN;
	ELSE
		//btn_UserGapStop:=FALSE;
		Error:=FALSE;
		ErrorId:=0;
		ErrorDescription:='';
	END_IF
	IF NOT inRange_UserTaperPositionNew THEN
		btn_UserGapStop:=TRUE;
		btn_UserGapMove:=FALSE;
		Error:=TRUE;
		ErrorId:=803;
		ErrorDescription:='target Taper Position out of range,please check';
		RETURN;
	ELSE
		//btn_UserGapStop:=FALSE;
		Error:=FALSE;
		ErrorId:=0;
		ErrorDescription:='';
	END_IF
	IF NOT inRange_UserTaperVelocityNew THEN
		btn_UserGapStop:=TRUE;
		btn_UserGapMove:=FALSE;
		Error:=TRUE;
		ErrorId:=804;
		ErrorDescription:='target Taper velocity out of range,please check';
		RETURN;
	ELSE
		//btn_UserGapStop:=FALSE;
		Error:=FALSE;
		ErrorId:=0;
		ErrorDescription:='';
	END_IF
END_IF

//
//运动过程中，监控目标位置速度
//
IF moveStatusAnyAxis THEN
	IF NOT inRange_UserGapPositionNew THEN
		btn_UserGapStop:=TRUE;
		Error:=TRUE;
		ErrorId:=805;
		ErrorDescription:='target Gap position out of range in moving process!';
		FB_PlcEmergencyStop();
	END_IF
	IF NOT inRange_UserGapVelocityNew THEN
		btn_UserGapStop:=TRUE;
		Error:=TRUE;
		ErrorId:=806;
		ErrorDescription:='target Gap velocity out of range in moving process!';
		FB_PlcEmergencyStop();
	END_IF
	IF NOT inRange_UserTaperPositionNew THEN
		btn_UserGapStop:=TRUE;
		Error:=TRUE;
		ErrorId:=807;
		ErrorDescription:='target Taper Position out of range in moving process!';
		FB_PlcEmergencyStop();
	END_IF
	IF NOT inRange_UserTaperVelocityNew THEN
		btn_UserGapStop:=TRUE;
		Error:=TRUE;
		ErrorId:=808;
		ErrorDescription:='target Taper velocity out of range in moving process!';
		FB_PlcEmergencyStop();
	END_IF
END_IF
//
//运动过程中，监控每一个轴的目标位置，目标位置若超出阈值，Emergency
//
IF moveStatusAnyAxis THEN
	IF NOT TaperOrNot THEN
		IF LeftTopLinPositionNew<min_UserLEProtectionGapPosition/2 OR LeftTopLinPositionNew>max_UserLEProtectionGapPosition/2 THEN
			btn_UserGapStop:=TRUE;
			Error:=TRUE;
			ErrorId:=809;
			ErrorDescription:='target LeftTop position out of range in moving process!';
			FB_PlcEmergencyStop();
		END_IF
		IF RightTopLinPositionNew<min_UserLEProtectionGapPosition/2 OR RightTopLinPositionNew>max_UserLEProtectionGapPosition/2 THEN
			btn_UserGapStop:=TRUE;
			Error:=TRUE;
			ErrorId:=810;
			ErrorDescription:='target RightTop velocity out of range in moving process!';
			FB_PlcEmergencyStop();
		END_IF
		IF LeftBottomLinPositionNew<min_UserLEProtectionGapPosition/2 OR LeftBottomLinPositionNew>max_UserLEProtectionGapPosition/2 THEN
			btn_UserGapStop:=TRUE;
			Error:=TRUE;
			ErrorId:=812;
			ErrorDescription:='target LeftBottom Position out of range in moving process!';
			FB_PlcEmergencyStop();
		END_IF
		IF RightBottomLinPositionNew<min_UserLEProtectionGapPosition/2 OR RightBottomLinPositionNew>max_UserLEProtectionGapPosition/2 THEN
			btn_UserGapStop:=TRUE;
			Error:=TRUE;
			ErrorId:=813;
			ErrorDescription:='target RightBottom Position out of range in moving process!';
			FB_PlcEmergencyStop();
		END_IF
		IF LeftInLinPositionNew<min_UserLEProtectionGapPosition/2 OR LeftInLinPositionNew>max_UserLEProtectionGapPosition/2 THEN
			btn_UserGapStop:=TRUE;
			Error:=TRUE;
			ErrorId:=809;
			ErrorDescription:='target LeftIn position out of range in moving process!';
			FB_PlcEmergencyStop();
		END_IF
		IF RightInLinPositionNew<min_UserLEProtectionGapPosition/2 OR RightInLinPositionNew>max_UserLEProtectionGapPosition/2 THEN
			btn_UserGapStop:=TRUE;
			Error:=TRUE;
			ErrorId:=810;
			ErrorDescription:='target RightIn velocity out of range in moving process!';
			FB_PlcEmergencyStop();
		END_IF
		IF LeftOutLinPositionNew<min_UserLEProtectionGapPosition/2 OR LeftOutLinPositionNew>max_UserLEProtectionGapPosition/2 THEN
			btn_UserGapStop:=TRUE;
			Error:=TRUE;
			ErrorId:=812;
			ErrorDescription:='target LeftOut Position out of range in moving process!';
			FB_PlcEmergencyStop();
		END_IF
		IF RightOutLinPositionNew<min_UserLEProtectionGapPosition/2 OR RightOutLinPositionNew>max_UserLEProtectionGapPosition/2 THEN
			btn_UserGapStop:=TRUE;
			Error:=TRUE;
			ErrorId:=813;
			ErrorDescription:='target RightOut Position out of range in moving process!';
			FB_PlcEmergencyStop();
		END_IF
	ELSE//Taper状态的保护
		;//Taper状态下，不用监控四轴位置，只需要监控目标Taper位置。在上面已经保护
	END_IF
END_IF
END_ACTION

ACTION A_GlobalChainProtection_EPS:
//硬线输入定义
Global_ChainProtection_EPS_In:=Global_ChainProtection_EPS_In1 AND Global_ChainProtection_EPS_In2;
//硬线输出定义
Global_ChainProtection_EPS_Out1:=Global_ChainProtection_EPS_Done;
Global_ChainProtection_EPS_Out2:=Global_ChainProtection_EPS_Done;
//总开关
IF NOT Global_ChainProtection_EPS_On THEN
	RETURN;
END_IF
//判断插入件状态，是否就位
//IF NOT IDControlReady THEN
//	Global_ChainProtection_EPS_Done:=FALSE;
//	Error:= TRUE;
//	ErrorID:= 1501;
//	ErrorDescription:='ID NOT READY!';
//	RETURN;
//END_IF
//判断储存环是否给出就位信号，暂时由参数表给出TRUE，最终将由IOC接受PV
IF 	NOT Global_ChainProtection_EPS_BeamLineReady THEN
	Global_ChainProtection_EPS_Done:=FALSE;
	Error:= TRUE;
	ErrorID:= 1503;
	ErrorDescription:='Global_ChainProtection_EPS_BeamLineReady NOT Ready';
	RETURN;
END_IF
//
//全局连锁保护程序开始
//
//0.检测到下降沿，触发
//1.判断电机是否在开启状态,没有就打开电源
//2.判断是否在Moving状态,若有就Stop
//3.将磁间隙打开到至最大阈值
//4.到位后给出反馈，且安全PLC触发
Global_ChainProtection_EPS_FTRIG(CLK:=Global_ChainProtection_EPS_In);
IF Global_ChainProtection_EPS_FTRIG.Q THEN
	Global_ChainProtection_EPS_Triggered:=TRUE;
END_IF
Global_ChainProtection_EPS_FTRIG_Manul(CLK:=Global_ChainProtection_EPS_ManualOperation);
IF Global_ChainProtection_EPS_FTRIG_Manul.Q THEN
	Global_ChainProtection_EPS_Triggered:=TRUE;
END_IF
IF Global_ChainProtection_EPS_Triggered THEN
	CASE Global_ChainProtection_EPS_State OF
		0://1.判断电机是否在开启状态,没有就打开电源
			IF st_Power=1 THEN
				Global_ChainProtection_EPS_State:=1;
			ELSE
				btn_PowerOn:=TRUE;
				IF btn_PowerOn THEN
					A_PowerOn();
				END_IF
			END_IF
		1://1.判断是否在谱学扫描模式，如果是，则切换回正常运动模式
			IF IsSSMotionMode THEN
				SS_Stop:=TRUE;
				IsSSMotionMode:=FALSE;
			END_IF
			Global_ChainProtection_EPS_State:=2;
		2://判断是否在taper，如果在taper,则判断是否在运动，如果是，则停止运动,0.5sh后，转入下一步
			IF TaperOrNot THEN
				IF moveStatusLeftTop OR moveStatusRightTop OR moveStatusLeftBottom OR moveStatusRightBottom 
					OR moveStatusLeftIn OR moveStatusRightIn OR moveStatusLeftOut OR moveStatusRightOut THEN
					btn_UserGapStop:=TRUE;
				ELSE
					Global_ChainProtection_EPS_TON_Stop2Move_InTaperMode(PT:=T#0.5S);
					Global_ChainProtection_EPS_TON_Stop2Move_InTaperMode.IN:=TRUE;
					IF Global_ChainProtection_EPS_TON_Stop2Move_InTaperMode.Q THEN
						TaperOrNot:=FALSE;//关闭taper模式
						Global_ChainProtection_EPS_State:=3;
					END_IF
				END_IF
			ELSE
				Global_ChainProtection_EPS_State:=3;
			END_IF
		3://3.判断是否在Moving状态,若有就Stop.Taper模式已处理完，此处开始走正常GAP开合逻辑
			IF moveStatusLeftTop OR moveStatusRightTop OR moveStatusLeftBottom OR moveStatusRightBottom 
					OR moveStatusLeftIn OR moveStatusRightIn OR moveStatusLeftOut OR moveStatusRightOut THEN
				btn_UserGapStop:=TRUE;
			ELSE
				Global_ChainProtection_EPS_TON_Stop2Move(PT:=T#0.5S);
				Global_ChainProtection_EPS_TON_Stop2Move.IN:=TRUE;
				IF Global_ChainProtection_EPS_TON_Stop2Move.Q THEN
					Global_ChainProtection_EPS_State:=4;
				END_IF
			END_IF
		4://当前磁间隙如何和最大磁间隙差别不大，不超过0.1，则直接保护
			IF ABS(UserGapPositionDisplay-Global_ChainProtection_EPS_MaxGapValue)<=0.1 THEN
				Global_ChainProtection_EPS_Done:=TRUE;
				Plc_EmergencyStop:=FALSE;	
				Error:=TRUE;
				ErrorID:=1506;
				ErrorDescription:='EPS Triggered,but ABS(UserGapPositionDisplay-Global_ChainProtection_EPS_MaxGapValue)<=0.1 ';	
			ELSE
				Global_ChainProtection_EPS_State:=5;
			END_IF
		5://5.将磁间隙打开到至最大阈值
			Global_ChainProtection_EPS_TON(PT:=INT_TO_TIME(LREAL_TO_INT(Global_ChainProtection_EPS_MaxGapValue/Global_ChainProtection_EPS_MoveVelocity+30))*1000);
			Global_ChainProtection_EPS_TON.IN:=TRUE;
			Global_ChainProtection_EPS_TON_Power2Move(PT:=T#0.1S);
			Global_ChainProtection_EPS_TON_Power2Move.IN:=TRUE;
			UserGapPositionNew:=Global_ChainProtection_EPS_MaxGapValue;
			UserGapVelocityNew:=Global_ChainProtection_EPS_MoveVelocity;
			btn_UserGapMove:=TRUE;
			IF Global_ChainProtection_EPS_TON_Power2Move.Q THEN
				IF FB_MOVE.BCGapDone THEN
					Global_ChainProtection_EPS_State:=88;
				END_IF
			END_IF
			IF Global_ChainProtection_EPS_TON.Q THEN//如果150s后，还没有运动到指定gap，则报错
				Global_ChainProtection_EPS_State:=-100;
			END_IF
		88://6.到位后给出反馈，且安全PLC触发
			Global_ChainProtection_EPS_Done:=TRUE;
			Plc_EmergencyStop:=FALSE;	
			Error:=TRUE;
			ErrorID:=1504;
			ErrorDescription:='Global_ChainProtection_EPS Triggered ';	
		-100:
			Global_ChainProtection_EPS_Done:=FALSE;
			Error:=TRUE;
			ErrorID:=1505;
			ErrorDescription:='NOT MOVING TO MAXGAP';
	END_CASE
END_IF

(*
//硬线输入定义
Global_ChainProtection_EPS_In:=Global_ChainProtection_EPS_In1 AND Global_ChainProtection_EPS_In2;
//硬线输出定义
Global_ChainProtection_EPS_Out1:=Global_ChainProtection_EPS_Done;
Global_ChainProtection_EPS_Out2:=Global_ChainProtection_EPS_Done;
//总开关
IF NOT Global_ChainProtection_EPS_On THEN
	RETURN;
END_IF
//判断插入件状态，是否就位
//IF NOT IDControlReady THEN
//	Global_ChainProtection_EPS_Done:=FALSE;
//	Error:= TRUE;
//	ErrorID:= 1501;
//	ErrorDescription:='ID NOT READY!';
//	RETURN;
//END_IF
//判断储存环是否给出就位信号，暂时由参数表给出TRUE，最终将由IOC接受PV
IF 	NOT Global_ChainProtection_EPS_BeamLineReady THEN
	Global_ChainProtection_EPS_Done:=FALSE;
	Error:= TRUE;
	ErrorID:= 1503;
	ErrorDescription:='Global_ChainProtection_EPS_BeamLineReady NOT Ready';
	RETURN;
END_IF
//
//全局连锁保护程序开始
//
//0.检测到下降沿，触发
//1.判断电机是否在开启状态,没有就打开电源
//2.判断是否在Moving状态,若有就Stop
//3.将磁间隙打开到至最大阈值
//4.到位后给出反馈，且安全PLC触发
Global_ChainProtection_EPS_FTRIG(CLK:=Global_ChainProtection_EPS_In);
IF Global_ChainProtection_EPS_FTRIG.Q THEN
	Global_ChainProtection_EPS_Triggered:=TRUE;
END_IF
Global_ChainProtection_EPS_FTRIG_Manul(CLK:=Global_ChainProtection_EPS_ManualOperation);
IF Global_ChainProtection_EPS_FTRIG_Manul.Q THEN
	Global_ChainProtection_EPS_Triggered:=TRUE;
END_IF
IF Global_ChainProtection_EPS_Triggered THEN
	CASE Global_ChainProtection_EPS_State OF
		0://1.判断电机是否在开启状态,没有就打开电源
			IF st_Power=1 THEN
				Global_ChainProtection_EPS_State:=1;
			ELSE
				btn_PowerOn:=TRUE;
				IF btn_PowerOn THEN
					A_PowerOn();
				END_IF
			END_IF
		1://1.判断是否在谱学扫描模式，如果是，则切换回正常运动模式
			IF IsSSMotionMode THEN
				SS_Stop:=TRUE;
				IsSSMotionMode:=FALSE;
			END_IF
			Global_ChainProtection_EPS_State:=2;
		2://判断是否在taper，如果在taper,则判断是否在运动，如果是，则停止运动,0.5sh后，转入下一步
			IF TaperOrNot THEN
				IF moveStatusLeftTop OR moveStatusRightTop OR moveStatusLeftBottom OR moveStatusRightBottom 
					OR moveStatusLeftIn OR moveStatusRightIn OR moveStatusLeftOut OR moveStatusRightOut THEN
					btn_UserGapStop:=TRUE;
				ELSE
					Global_ChainProtection_EPS_TON_Stop2Move_InTaperMode(PT:=T#0.5S);
					Global_ChainProtection_EPS_TON_Stop2Move_InTaperMode.IN:=TRUE;
					IF Global_ChainProtection_EPS_TON_Stop2Move_InTaperMode.Q THEN
						TaperOrNot:=FALSE;//关闭taper模式
						Global_ChainProtection_EPS_State:=3;
					END_IF
				END_IF
			ELSE
				Global_ChainProtection_EPS_State:=3;
			END_IF
		3://3.判断是否在Moving状态,若有就Stop.Taper模式已处理完，此处开始走正常GAP开合逻辑
			IF moveStatusLeftTop OR moveStatusRightTop OR moveStatusLeftBottom OR moveStatusRightBottom 
				OR moveStatusLeftIn OR moveStatusRightIn OR moveStatusLeftOut OR moveStatusRightOut THEN
				btn_UserGapStop:=TRUE;
			ELSE
				Global_ChainProtection_EPS_TON_Stop2Move(PT:=T#0.5S);
				Global_ChainProtection_EPS_TON_Stop2Move.IN:=TRUE;
				IF Global_ChainProtection_EPS_TON_Stop2Move.Q THEN
					Global_ChainProtection_EPS_State:=4;
				END_IF
			END_IF
		4://4.将磁间隙打开到至最大阈值
			Global_ChainProtection_EPS_TON(PT:=INT_TO_TIME(LREAL_TO_INT(Global_ChainProtection_EPS_MaxGapValue/Global_ChainProtection_EPS_MoveVelocity+30))*1000);
			Global_ChainProtection_EPS_TON.IN:=TRUE;
			Global_ChainProtection_EPS_TON_Power2Move(PT:=T#0.1S);
			Global_ChainProtection_EPS_TON_Power2Move.IN:=TRUE;
			UserGapPositionNew:=Global_ChainProtection_EPS_MaxGapValue;
			UserGapVelocityNew:=Global_ChainProtection_EPS_MoveVelocity;
			btn_UserGapMove:=TRUE;
			IF Global_ChainProtection_EPS_TON_Power2Move.Q THEN
				IF FB_MOVE.BCGapDone THEN
					Global_ChainProtection_EPS_State:=88;
				END_IF
			END_IF
			IF Global_ChainProtection_EPS_TON.Q THEN//如果150s后，还没有运动到指定gap，则报错
				Global_ChainProtection_EPS_State:=-100;
			END_IF
		88://4.到位后给出反馈，且安全PLC触发
			Global_ChainProtection_EPS_Done:=TRUE;
			Plc_EmergencyStop:=FALSE;	
			Error:=TRUE;
			ErrorID:=1504;
			ErrorDescription:='Global_ChainProtection_EPS Triggered ';	
		-100:
			Global_ChainProtection_EPS_Done:=FALSE;
			Error:=TRUE;
			ErrorID:=1505;
			ErrorDescription:='NOT MOVING TO MAXGAP';
	END_CASE
END_IF
*)
END_ACTION

ACTION A_GlobalChainProtection_MPS:
//硬线输入定义
Global_ChainProtection_MPS_In:=Global_ChainProtection_MPS_In1 AND Global_ChainProtection_MPS_In2;
//硬线输出定义
Global_ChainProtection_MPS_Out1:=Global_ChainProtection_MPS_Done;
Global_ChainProtection_MPS_Out2:=Global_ChainProtection_MPS_Done;
//总开关
IF NOT Global_ChainProtection_MPS_On THEN
	RETURN;
END_IF
//判断插入件状态，是否就位
//IF NOT IDControlReady THEN
//	Global_ChainProtection_MPS_Done:=FALSE;
//	Error:= TRUE;
//	ErrorID:= 1401;
//	ErrorDescription:='ID NOT READY!';
//	RETURN;
//END_IF
//判断储存环是否给出就位信号，暂时由参数表给出TRUE，最终将由IOC接受PV
IF 	NOT Global_ChainProtection_MPS_StorageRingReady THEN
	Global_ChainProtection_MPS_Done:=FALSE;
	Error:= TRUE;
	ErrorID:= 1403;
	ErrorDescription:='StorageRingChainProtection NOT Ready';
	RETURN;
END_IF
//
//全局连锁保护程序开始
//
//0.检测到下降沿，触发
//1.判断电机是否在开启状态,没有就打开电源
//2.判断是否在Moving状态,若有就Stop
//3.将磁间隙打开到至最大阈值
//4.到位后给出反馈，且安全PLC触发
Global_ChainProtection_MPS_FTRIG(CLK:=Global_ChainProtection_MPS_In);
IF Global_ChainProtection_MPS_FTRIG.Q THEN
	Global_ChainProtection_MPS_Triggered:=TRUE;
END_IF
Global_ChainProtection_MPS_FTRIG_Manul(CLK:=Global_ChainProtection_MPS_ManualOperation);
IF Global_ChainProtection_MPS_FTRIG_Manul.Q THEN
	Global_ChainProtection_MPS_Triggered:=TRUE;
END_IF
IF Global_ChainProtection_MPS_Triggered THEN
	CASE Global_ChainProtection_MPS_State OF
		0://1.判断电机是否在开启状态,没有就打开电源
			IF st_Power=1 THEN
				Global_ChainProtection_MPS_State:=1;
			ELSE
				btn_PowerOn:=TRUE;
				IF btn_PowerOn THEN
					A_PowerOn();
				END_IF
			END_IF
		1://1.判断是否在谱学扫描模式，如果是，则切换回正常运动模式
			IF IsSSMotionMode THEN
				SS_Stop:=TRUE;
				IsSSMotionMode:=FALSE;
			END_IF
			Global_ChainProtection_MPS_State:=2;
		2://判断是否在taper，如果在taper,则判断是否在运动，如果是，则停止运动,0.5sh后，转入下一步
			IF TaperOrNot THEN
				IF moveStatusLeftTop OR moveStatusRightTop OR moveStatusLeftBottom OR moveStatusRightBottom 
					OR moveStatusLeftIn OR moveStatusRightIn OR moveStatusLeftOut OR moveStatusRightOut THEN
					btn_UserGapStop:=TRUE;
				ELSE
					Global_ChainProtection_MPS_TON_Stop2Move_InTaperMode(PT:=T#0.5S);
					Global_ChainProtection_MPS_TON_Stop2Move_InTaperMode.IN:=TRUE;
					IF Global_ChainProtection_MPS_TON_Stop2Move_InTaperMode.Q THEN
						TaperOrNot:=FALSE;//关闭taper模式
						Global_ChainProtection_MPS_State:=3;
					END_IF
				END_IF
			ELSE
				Global_ChainProtection_MPS_State:=3;
			END_IF
		3://3.判断是否在Moving状态,若有就Stop.Taper模式已处理完，此处开始走正常GAP开合逻辑
			IF moveStatusLeftTop OR moveStatusRightTop OR moveStatusLeftBottom OR moveStatusRightBottom 
					OR moveStatusLeftIn OR moveStatusRightIn OR moveStatusLeftOut OR moveStatusRightOut THEN
					btn_UserGapStop:=TRUE;
				ELSE
				Global_ChainProtection_MPS_TON_Stop2Move(PT:=T#0.5S);
				Global_ChainProtection_MPS_TON_Stop2Move.IN:=TRUE;
				IF Global_ChainProtection_MPS_TON_Stop2Move.Q THEN
					Global_ChainProtection_MPS_State:=4;
				END_IF
			END_IF
		4://当前磁间隙如何和最大磁间隙差别不大，不超过0.1，则直接保护
			IF ABS(UserGapPositionDisplay-Global_ChainProtection_MPS_MaxGapValue)<=0.1 THEN
				Global_ChainProtection_MPS_Done:=TRUE;
				Plc_EmergencyStop:=FALSE;	
				Error:=TRUE;
				ErrorID:=1406;
				ErrorDescription:='MPS Triggered,but ABS(UserGapPositionDisplay-Global_ChainProtection_MPS_MaxGapValue)<=0.1 ';	
			ELSE
				Global_ChainProtection_MPS_State:=5;
			END_IF
		5://5.将磁间隙打开到至最大阈值
			Global_ChainProtection_MPS_TON(PT:=INT_TO_TIME(LREAL_TO_INT(Global_ChainProtection_MPS_MaxGapValue/Global_ChainProtection_MPS_MoveVelocity+30))*1000);
			Global_ChainProtection_MPS_TON.IN:=TRUE;
			Global_ChainProtection_MPS_TON_Power2Move(PT:=T#0.1S);
			Global_ChainProtection_MPS_TON_Power2Move.IN:=TRUE;
			UserGapPositionNew:=Global_ChainProtection_MPS_MaxGapValue;
			UserGapVelocityNew:=Global_ChainProtection_MPS_MoveVelocity;
			btn_UserGapMove:=TRUE;
			IF Global_ChainProtection_MPS_TON_Power2Move.Q THEN
				IF FB_MOVE.BCGapDone THEN
					Global_ChainProtection_MPS_State:=88;
				END_IF
			END_IF
			IF Global_ChainProtection_MPS_TON.Q THEN//如果150s后，还没有运动到指定gap，则报错
				Global_ChainProtection_MPS_State:=-100;
			END_IF
		88://6.到位后给出反馈，且安全PLC触发
			Global_ChainProtection_MPS_Done:=TRUE;
			Plc_EmergencyStop:=FALSE;	
			Error:=TRUE;
			ErrorID:=1404;
			ErrorDescription:='Global_ChainProtection_MPS Triggered ';	
		-100:
			Global_ChainProtection_MPS_Done:=FALSE;
			Error:=TRUE;
			ErrorID:=1405;
			ErrorDescription:='NOT MOVING TO MAXGAP';
	END_CASE
END_IF


(*
//硬线输入定义
Global_ChainProtection_MPS_In:=Global_ChainProtection_MPS_In1 AND Global_ChainProtection_MPS_In2;
//硬线输出定义
Global_ChainProtection_MPS_Out1:=Global_ChainProtection_MPS_Done;
Global_ChainProtection_MPS_Out2:=Global_ChainProtection_MPS_Done;
//总开关
IF NOT Global_ChainProtection_MPS_On THEN
	RETURN;
END_IF
//判断插入件状态，是否就位
//IF NOT IDControlReady THEN
//	Global_ChainProtection_MPS_Done:=FALSE;
//	Error:= TRUE;
//	ErrorID:= 1401;
//	ErrorDescription:='ID NOT READY!';
//	RETURN;
//END_IF
//判断储存环是否给出就位信号，暂时由参数表给出TRUE，最终将由IOC接受PV
IF 	NOT Global_ChainProtection_MPS_StorageRingReady THEN
	Global_ChainProtection_MPS_Done:=FALSE;
	Error:= TRUE;
	ErrorID:= 1403;
	ErrorDescription:='StorageRingChainProtection NOT Ready';
	RETURN;
END_IF
//
//全局连锁保护程序开始
//
//0.检测到下降沿，触发
//1.判断电机是否在开启状态,没有就打开电源
//2.判断是否在Moving状态,若有就Stop
//3.将磁间隙打开到至最大阈值
//4.到位后给出反馈，且安全PLC触发
Global_ChainProtection_MPS_FTRIG(CLK:=Global_ChainProtection_MPS_In);
IF Global_ChainProtection_MPS_FTRIG.Q THEN
	Global_ChainProtection_MPS_Triggered:=TRUE;
END_IF
Global_ChainProtection_MPS_FTRIG_Manul(CLK:=Global_ChainProtection_MPS_ManualOperation);
IF Global_ChainProtection_MPS_FTRIG_Manul.Q THEN
	Global_ChainProtection_MPS_Triggered:=TRUE;
END_IF
IF Global_ChainProtection_MPS_Triggered THEN
	CASE Global_ChainProtection_MPS_State OF
		0://1.判断电机是否在开启状态,没有就打开电源
			IF st_Power=1 THEN
				Global_ChainProtection_MPS_State:=1;
			ELSE
				btn_PowerOn:=TRUE;
				IF btn_PowerOn THEN
					A_PowerOn();
				END_IF
			END_IF
		1://1.判断是否在谱学扫描模式，如果是，则切换回正常运动模式
			IF IsSSMotionMode THEN
				SS_Stop:=TRUE;
				IsSSMotionMode:=FALSE;
			END_IF
			Global_ChainProtection_MPS_State:=2;
		2://判断是否在taper，如果在taper,则判断是否在运动，如果是，则停止运动,0.5sh后，转入下一步
			IF TaperOrNot THEN
				IF moveStatusLeftTop OR moveStatusRightTop OR moveStatusLeftBottom OR moveStatusRightBottom 
					OR moveStatusLeftIn OR moveStatusRightIn OR moveStatusLeftOut OR moveStatusRightOut THEN
					btn_UserGapStop:=TRUE;
				ELSE
					Global_ChainProtection_MPS_TON_Stop2Move_InTaperMode(PT:=T#0.5S);
					Global_ChainProtection_MPS_TON_Stop2Move_InTaperMode.IN:=TRUE;
					IF Global_ChainProtection_MPS_TON_Stop2Move_InTaperMode.Q THEN
						TaperOrNot:=FALSE;//关闭taper模式
						Global_ChainProtection_MPS_State:=3;
					END_IF
				END_IF
			ELSE
				Global_ChainProtection_MPS_State:=3;
			END_IF
		3://3.判断是否在Moving状态,若有就Stop.Taper模式已处理完，此处开始走正常GAP开合逻辑
			IF moveStatusLeftTop OR moveStatusRightTop OR moveStatusLeftBottom OR moveStatusRightBottom 
					OR moveStatusLeftIn OR moveStatusRightIn OR moveStatusLeftOut OR moveStatusRightOut THEN
				btn_UserGapStop:=TRUE;
			ELSE
				Global_ChainProtection_MPS_TON_Stop2Move(PT:=T#0.5S);
				Global_ChainProtection_MPS_TON_Stop2Move.IN:=TRUE;
				IF Global_ChainProtection_MPS_TON_Stop2Move.Q THEN
					Global_ChainProtection_MPS_State:=4;
				END_IF
			END_IF
		4://4.将磁间隙打开到至最大阈值
			Global_ChainProtection_MPS_TON(PT:=INT_TO_TIME(LREAL_TO_INT(Global_ChainProtection_MPS_MaxGapValue/Global_ChainProtection_MPS_MoveVelocity+30))*1000);
			Global_ChainProtection_MPS_TON.IN:=TRUE;
			Global_ChainProtection_MPS_TON_Power2Move(PT:=T#0.1S);
			Global_ChainProtection_MPS_TON_Power2Move.IN:=TRUE;
			UserGapPositionNew:=Global_ChainProtection_MPS_MaxGapValue;
			UserGapVelocityNew:=Global_ChainProtection_MPS_MoveVelocity;
			btn_UserGapMove:=TRUE;
			IF Global_ChainProtection_MPS_TON_Power2Move.Q THEN
				IF FB_MOVE.BCGapDone THEN
					Global_ChainProtection_MPS_State:=88;
				END_IF
			END_IF
			IF Global_ChainProtection_MPS_TON.Q THEN//如果150s后，还没有运动到指定gap，则报错
				Global_ChainProtection_MPS_State:=-100;
			END_IF
		88://4.到位后给出反馈，且安全PLC触发
			Global_ChainProtection_MPS_Done:=TRUE;
			Plc_EmergencyStop:=FALSE;	
			Error:=TRUE;
			ErrorID:=1404;
			ErrorDescription:='Global_ChainProtection_MPS Triggered ';	
		-100:
			Global_ChainProtection_MPS_Done:=FALSE;
			Error:=TRUE;
			ErrorID:=1405;
			ErrorDescription:='NOT MOVING TO MAXGAP';
	END_CASE
END_IF
*)
END_ACTION

ACTION A_InitCompensationData:
(*补偿开始*)
IF USE_SingleAxis_Compensation THEN
	//
	//1.目标位置解算
	//
	(*通过补偿表解算四轴目标位置*)
	//左轴位置由Gap定，右轴位置由右gap定。右gap值=左gap+taper。taper模式和非taper模式一样，非taper模式只是一种特例存在
	//左轴目标位置解算
	IF NOT TaperOrNot THEN
		UserTaperPositionNew:=0;
		//UserTaperPositionDisplay:=0;
	END_IF
	UserRightGapPositionNew:=UserGapPositionNew+UserTaperPositionNew;
	//左轴目标位置解算
	FOR	i:= 1 TO 17 DO
			IF UserGapPositionNew/2<M_Compensation[i+1].Encoder AND UserGapPositionNew/2>=M_Compensation[i].Encoder THEN
				IF i<>18 THEN
					LeftTopLinPositionNew:=(((UserGapPositionNew/2-M_Compensation[i].Encoder)*(M_Compensation[i+1].LeftTop-M_Compensation[i].LeftTop))
							/(M_Compensation[i+1].Encoder-M_Compensation[i].Encoder))+M_Compensation[i].LeftTop;
					LeftBottomLinPositionNew:=(((UserGapPositionNew/2-M_Compensation[i].Encoder)*(M_Compensation[i+1].LeftBottom-M_Compensation[i].LeftBottom))
							/(M_Compensation[i+1].Encoder-M_Compensation[i].Encoder))+M_Compensation[i].LeftBottom;
					LeftInLinPositionNew:=(((UserGapPositionNew/2-M_Compensation[i].Encoder)*(M_Compensation[i+1].LeftIn-M_Compensation[i].LeftIn))
							/(M_Compensation[i+1].Encoder-M_Compensation[i].Encoder))+M_Compensation[i].LeftIn;
					LeftOutLinPositionNew:=(((UserGapPositionNew/2-M_Compensation[i].Encoder)*(M_Compensation[i+1].LeftOut-M_Compensation[i].LeftOut))
							/(M_Compensation[i+1].Encoder-M_Compensation[i].Encoder))+M_Compensation[i].LeftOut;
					M_CompensationNumber:=i;
					InitCompensationDatasDone:=TRUE;
				ELSIF i=18 AND UserGapPositionNew/2=M_Compensation[i].Encoder THEN		(*Gap=14µÄÌØÊâÇé¿ö*)
					(**)
					LeftTopLinPositionNew:=M_Compensation[i].LeftTop;
					LeftBottomLinPositionNew:=M_Compensation[i].LeftBottom;
					LeftInLinPositionNew:=M_Compensation[i].LeftIn;
					LeftOutLinPositionNew:=M_Compensation[i].LeftOut;
					M_CompensationNumber:=i;
					InitCompensationDatasDone:=TRUE;
				ELSE
					LeftTopLinPositionNew:=UserGapPositionNew/2;
					LeftBottomLinPositionNew:=UserGapPositionNew/2;
					LeftInLinPositionNew:=UserGapPositionNew/2;
					LeftOutLinPositionNew:=UserGapPositionNew/2;
					M_CompensationNumber:=i;
					InitCompensationDatasDone:=TRUE;
				END_IF
			END_IF
	END_FOR
	//右轴目标位置解算
	FOR	j:= 1 TO 17 DO
		IF UserRightGapPositionNew/2<M_Compensation[j+1].Encoder AND UserRightGapPositionNew/2>=M_Compensation[j].Encoder THEN
			IF j<>18 THEN
				RightTopLinPositionNew:=(((UserRightGapPositionNew/2-M_Compensation[j].Encoder)*(M_Compensation[j+1].RightTop-M_Compensation[j].RightTop))
						/(M_Compensation[j+1].Encoder-M_Compensation[j].Encoder))+M_Compensation[j].RightTop;
				RightBottomLinPositionNew:=(((UserRightGapPositionNew/2-M_Compensation[j].Encoder)*(M_Compensation[j+1].RightBottom-M_Compensation[j].RightBottom))
						/(M_Compensation[j+1].Encoder-M_Compensation[j].Encoder))+M_Compensation[j].RightBottom;
				RightInLinPositionNew:=(((UserRightGapPositionNew/2-M_Compensation[j].Encoder)*(M_Compensation[j+1].RightIn-M_Compensation[j].RightIn))
						/(M_Compensation[j+1].Encoder-M_Compensation[j].Encoder))+M_Compensation[j].RightIn;
				RightOutLinPositionNew:=(((UserRightGapPositionNew/2-M_Compensation[j].Encoder)*(M_Compensation[j+1].RightOut-M_Compensation[j].RightOut))
						/(M_Compensation[j+1].Encoder-M_Compensation[j].Encoder))+M_Compensation[j].RightOut;
				M_CompensationNumber:=j;
				InitCompensationDatasDone:=TRUE;
			ELSIF j=18 AND UserRightGapPositionNew/2=M_Compensation[i].Encoder THEN		(*Gap=14µÄÌØÊâÇé¿ö*)
				(**)
				RightTopLinPositionNew:=M_Compensation[i].RightTop;
				RightBottomLinPositionNew:=M_Compensation[i].RightBottom;
				RightInLinPositionNew:=M_Compensation[i].RightIn;
				RightOutLinPositionNew:=M_Compensation[i].RightOut;
				M_CompensationNumber:=j;
				InitCompensationDatasDone:=TRUE;
			ELSE
				RightTopLinPositionNew:=UserGapPositionNew/2;
				RightBottomLinPositionNew:=UserGapPositionNew/2;
				RightInLinPositionNew:=UserGapPositionNew/2;
				RightOutLinPositionNew:=UserGapPositionNew/2;
				M_CompensationNumber:=j;
				InitCompensationDatasDone:=TRUE;
			END_IF
		END_IF
	END_FOR
	//
	//2.不论taper还是非taper模式，左轴gap都有左轴发推算，右轴gap由右轴反推算。taper为右gap-左gap
	//
	//左轴显示位置反结算
	FOR k:= 1 TO 17 DO
			IF Pos_LeftTopLin<M_Compensation[k+1].LeftTop AND Pos_LeftTopLin>=M_Compensation[k].LeftTop THEN
				UserGapPositionDisplay_FromLeftTop:=2*(((Pos_LeftTopLin-M_Compensation[k].LeftTop)*(M_Compensation[k+1].Encoder-M_Compensation[k].Encoder))
											/(M_Compensation[k+1].LeftTop-M_Compensation[k].LeftTop)+M_Compensation[k].Encoder);
				UserGapPositionDisplay_FromLeftBottom:=2*(((Pos_LeftBottomLin-M_Compensation[k].LeftBottom)*(M_Compensation[k+1].Encoder-M_Compensation[k].Encoder))
											/(M_Compensation[k+1].LeftBottom-M_Compensation[k].LeftBottom)+M_Compensation[k].Encoder);									
				UserGapPositionDisplay_FromLeftIn:=2*(((Pos_LeftInLin-M_Compensation[k].LeftIn)*(M_Compensation[k+1].Encoder-M_Compensation[k].Encoder))
											/(M_Compensation[k+1].LeftIn-M_Compensation[k].LeftIn)+M_Compensation[k].Encoder);
				UserGapPositionDisplay_FromLeftOut:=2*(((Pos_LeftOutLin-M_Compensation[k].LeftOut)*(M_Compensation[k+1].Encoder-M_Compensation[k].Encoder))
											/(M_Compensation[k+1].LeftOut-M_Compensation[k].LeftOut)+M_Compensation[k].Encoder);
				UserGapPositionDisplay:=DINT_TO_LREAL(LREAL_TO_DINT(((UserGapPositionDisplay_FromLeftTop+UserGapPositionDisplay_FromLeftBottom
																	+UserGapPositionDisplay_FromLeftIn+UserGapPositionDisplay_FromLeftOut)/4)*100000))/100000;
			END_IF
	END_FOR
	//右轴显示位置反结算
	FOR m:= 1 TO 17 DO
			IF Pos_RightTopLin<M_Compensation[m+1].RightTop AND Pos_RightTopLin>=M_Compensation[m].RightTop THEN
				UserRightGapPositionDisplay_FromRightTop:=2*(((Pos_RightTopLin-M_Compensation[m].RightTop)*(M_Compensation[m+1].Encoder-M_Compensation[m].Encoder))
											/(M_Compensation[m+1].RightTop-M_Compensation[m].RightTop)+M_Compensation[m].Encoder);
				UserRightGapPositionDisplay_FromRightBottom:=2*(((Pos_RightBottomLin-M_Compensation[m].RightBottom)*(M_Compensation[m+1].Encoder-M_Compensation[m].Encoder))
											/(M_Compensation[m+1].RightBottom-M_Compensation[m].RightBottom)+M_Compensation[m].Encoder);									
				UserRightGapPositionDisplay_FromRightIn:=2*(((Pos_RightInLin-M_Compensation[m].RightIn)*(M_Compensation[m+1].Encoder-M_Compensation[m].Encoder))
											/(M_Compensation[m+1].RightIn-M_Compensation[m].RightIn)+M_Compensation[m].Encoder);
				UserRightGapPositionDisplay_FromRightOut:=2*(((Pos_RightOutLin-M_Compensation[m].RightOut)*(M_Compensation[m+1].Encoder-M_Compensation[m].Encoder))
											/(M_Compensation[m+1].RightOut-M_Compensation[m].RightOut)+M_Compensation[m].Encoder);
				UserRightGapPositionDisplay:=DINT_TO_LREAL(LREAL_TO_DINT(((UserRightGapPositionDisplay_FromRightTop+UserRightGapPositionDisplay_FromRightBottom
												+UserRightGapPositionDisplay_FromRightIn+UserRightGapPositionDisplay_FromRightOut)/4)*100000))/100000;
			END_IF
	END_FOR
		IF TaperOrNot OR (Global_ChainProtection_MPS_Triggered OR Global_ChainProtection_EPS_Triggered)  THEN//安全联锁触发时，需要UserTaperPositionDisplay作为A_MonitoringAllAxis的保护
			UserTaperPositionDisplay:=DINT_TO_LREAL(LREAL_TO_DINT((UserRightGapPositionDisplay-UserGapPositionDisplay)*100000))/100000;
		UserTaperVelocityDisplay:=DINT_TO_LREAL(LREAL_TO_DINT((Velo_RightTopLin+Velo_RightBottomLin+Velo_RightInLin+Velo_RightOutLin)/4*100000))/100000;
	END_IF

	(*速度可以不用解算，直接用即可*)
	LeftTopLinVelocityDisplay:=Velo_LeftTopLin;
	RightTopLinVelocityDisplay:=Velo_RightTopLin;
	LeftBottomLinVelocityDisplay:=Velo_LeftBottomLin;
	RightBottomLinVelocityDisplay:=Velo_RightBottomLin;
	LeftInLinVelocityDisplay:=Velo_LeftInLin;
	RightInLinVelocityDisplay:=Velo_RightInLin;
	LeftOutLinVelocityDisplay:=Velo_LeftOutLin;
	RightOutLinVelocityDisplay:=Velo_RightOutLin;
	//Gap velocity
	UserGapVelocityDisplay:=DINT_TO_LREAL(LREAL_TO_DINT(((LeftTopLinVelocityDisplay+RightTopLinVelocityDisplay+
	LeftBottomLinVelocityDisplay+RightBottomLinVelocityDisplay+
	LeftInLinVelocityDisplay+RightInLinVelocityDisplay+
	LeftOutLinVelocityDisplay+RightOutLinVelocityDisplay)/4)*100000))/100000;

	(*解算单轴位置后，核验并做保护*)
	IF ABS(LeftTopLinPositionNew-UserGapPositionNew/2)>Threshold_motorsTargetPosCalculate THEN
		ErrorID:=1601;
		Error:=TRUE;
		ErrorDescription:='LeftTop Threshold_motorsTargetPosCalculate';
		FB_PlcEmergencyStop();
	END_IF
	//注意右轴解算以UserRightGapPositionNew为基准，考虑到taper
	IF ABS(RightTopLinPositionNew-UserRightGapPositionNew/2)>Threshold_motorsTargetPosCalculate THEN
		ErrorID:=1602;
		Error:=TRUE;
		ErrorDescription:='RightTop Threshold_motorsTargetPosCalculate';
		FB_PlcEmergencyStop();
	END_IF
	IF ABS(LeftBottomLinPositionNew-UserGapPositionNew/2)>Threshold_motorsTargetPosCalculate THEN
		ErrorID:=1603;
		Error:=TRUE;
		ErrorDescription:='LeftBottom Threshold_motorsTargetPosCalculate';
		FB_PlcEmergencyStop();
	END_IF
	//注意右轴解算以UserRightGapPositionNew为基准，考虑到taper
	IF ABS(RightBottomLinPositionNew-UserRightGapPositionNew/2)>Threshold_motorsTargetPosCalculate THEN
		ErrorID:=1604;
		Error:=TRUE;
		ErrorDescription:='RightBottom Threshold_motorsTargetPosCalculate';
		FB_PlcEmergencyStop();
	END_IF
	IF ABS(LeftInLinPositionNew-UserGapPositionNew/2)>Threshold_motorsTargetPosCalculate THEN
		ErrorID:=1605;
		Error:=TRUE;
		ErrorDescription:='LeftIn Threshold_motorsTargetPosCalculate';
		FB_PlcEmergencyStop();
	END_IF
	IF ABS(RightInLinPositionNew-UserRightGapPositionNew/2)>Threshold_motorsTargetPosCalculate THEN
		ErrorID:=1606;
		Error:=TRUE;
		ErrorDescription:='RightIn Threshold_motorsTargetPosCalculate';
		FB_PlcEmergencyStop();
	END_IF
	IF ABS(LeftOutLinPositionNew-UserGapPositionNew/2)>Threshold_motorsTargetPosCalculate THEN
		ErrorID:=1607;
		Error:=TRUE;
		ErrorDescription:='LeftOut Threshold_motorsTargetPosCalculate';
		FB_PlcEmergencyStop();
	END_IF
	IF ABS(RightOutLinPositionNew-UserRightGapPositionNew/2)>Threshold_motorsTargetPosCalculate THEN
		ErrorID:=1608;
		Error:=TRUE;
		ErrorDescription:='RightOut Threshold_motorsTargetPosCalculate';
		FB_PlcEmergencyStop();
	END_IF
END_IF
END_ACTION

ACTION A_MonitoringAllAxis:
(****************************************************************
NAME:			A_MonitoringAllAxis
DATA:			2018.1.9
VERSION:		1.0.0
DESCRIPTION:	
				Ã¿´ÎÑ­»·¾ùÖ´ÐÐÖáÎ»ÖÃºÍÖáÔË¶¯µÄ¼ì²é
				2.4Öá¹âÕ¤³ßÎ»ÖÃ¡¢ËÙ¶È¶Ô±È¼ì²é
HISTORY:
				2017.1.9		NEW

***************************************************************)

(*************************************************************************************2.4Öá¹âÕ¤³ßÎ»ÖÃ¡¢ËÙ¶È¶Ô±È¼ì²é**********************************************************************)
IF  st_Power<>0 THEN
CASE moni_State OF
(*Top Î»ÖÃºÍËÙ¶È±È¶Ô*)
0:
		//实际(*Position*)
		(*Top*)
		Diff_UserTopPos_actual:=ABS(Pos_leftTopLin-Pos_RightTopLin);
		(*Bottom*)
		Diff_UserBottomPos_actual:=ABS(Pos_LeftBottomLin-Pos_RightBottomLin);
		(*TBLeft*)
		Diff_UserTBLeftPos_actual:=ABS(Pos_LeftTopLin-Pos_LeftBottomLin);
		(*TBRight*)
		Diff_UserTBRightPos_actual:=ABS(Pos_RightTopLin-Pos_RightBottomLin);
		(*In*)
		Diff_UserInPos_actual:=ABS(Pos_leftInLin-Pos_RightInLin);
		(*Out*)
		Diff_UserOutPos_actual:=ABS(Pos_LeftOutLin-Pos_RightOutLin);
		(*IOLeft*)
		Diff_UserIOLeftPos_actual:=ABS(Pos_LeftInLin-Pos_LeftOutLin);
		(*IORight*)
		Diff_UserIORightPos_actual:=ABS(Pos_RightInLin-Pos_RightOutLin);
		(*Velocity*)
		(*Top*)
		Diff_UserTopVelo_actual:=ABS(Velo_leftTopLin-Velo_RightTopLin);
		(*Bottom*)
		Diff_UserBottomVelo_actual:=ABS(Velo_LeftBottomLin-Velo_RightBottomLin);
		(*TBLeft*)
		Diff_UserTBLeftVelo_actual:=ABS(Velo_LeftTopLin-Velo_LeftBottomLin);
		(*TBRight*)
		Diff_UserTBRightVelo_actual:=ABS(Velo_RightTopLin-Velo_RightBottomLin);
		(*In*)
		Diff_UserInVelo_actual:=ABS(Velo_leftInLin-Velo_RightInLin);
		(*Out*)
		Diff_UserOutVelo_actual:=ABS(Velo_LeftOutLin-Velo_RightOutLin);
		(*IOLeft*)
		Diff_UserIOLeftVelo_actual:=ABS(Velo_LeftInLin-Velo_LeftOutLin);
		(*IORight*)
		Diff_UserIORightVelo_actual:=ABS(Velo_RightInLin-Velo_RightOutLin);
		//阈值
		Threshold_UserTopPos_PLC:=Threshold_UserTopPos+UserTaperPositionDisplay;//Top位置误差=gap运动细微误差+目标taper位置
		Threshold_UserTopVelo_PLC:=Threshold_UserTopVelo+ABS(UserGapVelocityDisplay);//Top速度误差=gap运动细微误差+gap目标速度。因为可能出现一个轴运动完了，另一个轴还在运动的情况
		Threshold_UserBottomPos_PLC:=Threshold_UserBottomPos+UserTaperPositionDisplay;//Bottom同上
		Threshold_UserBottomVelo_PLC:=Threshold_UserBottomVelo+ABS(UserGapVelocityDisplay);//Bottom同上
		Threshold_UserTBLeftPos_PLC:=Threshold_UserTBLeftPos+UserTaperPositionDisplay;
		Threshold_UserTBLeftVelo_PLC:=Threshold_UserTBLeftVelo+ABS(UserGapVelocityDisplay);
		Threshold_UserTBRightPos_PLC:=Threshold_UserTBRightPos+UserTaperPositionDisplay;
		Threshold_UserTBRightVelo_PLC:=Threshold_UserTBRightVelo+ABS(UserGapVelocityDisplay);
		//
		
		Threshold_UserInPos_PLC:=Threshold_UserInPos+UserTaperPositionDisplay;//Top位置误差=gap运动细微误差+目标taper位置
		Threshold_UserInVelo_PLC:=Threshold_UserInVelo+ABS(UserGapVelocityDisplay);//Top速度误差=gap运动细微误差+gap目标速度。因为可能出现一个轴运动完了，另一个轴还在运动的情况
		Threshold_UserOutPos_PLC:=Threshold_UserOutPos+UserTaperPositionDisplay;//Bottom同上
		Threshold_UserOutVelo_PLC:=Threshold_UserOutVelo+ABS(UserGapVelocityDisplay);//Bottom同上
		Threshold_UserIOLeftPos_PLC:=Threshold_UserIOLeftPos+UserTaperPositionDisplay;
		Threshold_UserIOLeftVelo_PLC:=Threshold_UserIOLeftVelo+ABS(UserGapVelocityDisplay);
		Threshold_UserIORightPos_PLC:=Threshold_UserIORightPos+UserTaperPositionDisplay;
		Threshold_UserIORightVelo_PLC:=Threshold_UserIORightVelo+ABS(UserGapVelocityDisplay);
		//比较
		IF Diff_UserTopPos_actual >Threshold_UserTopPos_PLC THEN
				Error:=TRUE;
				ErrorID:=601;
				ErrorDescription:='Diff_UserTopPos_actual >Threshold_UserTopPos_PLC';
				moni_State:=-100;
		ELSIF Diff_UserTopVelo_actual>Threshold_UserTopVelo_PLC  THEN
				Error:=TRUE;
				ErrorID:=602;
				ErrorDescription:='Diff_UserTopVelo_actual>Threshold_UserTopVelo_PLC';
				moni_State:=-100;
		(*Bottom Î»ÖÃºÍËÙ¶È±È¶Ô*)
		ELSIF Diff_UserBottomPos_actual>Threshold_UserBottomPos_PLC THEN
				Error:=TRUE;
				ErrorID:=603;
				ErrorDescription:='Diff_UserBottomPos_actual>Threshold_UserBottomPos_PLC';
				moni_State:=-100;
		ELSIF Diff_UserBottomVelo_actual>Threshold_UserBottomVelo_PLC  THEN
				Error:=TRUE;
				ErrorID:=604;
				ErrorDescription:='Diff_UserBottomVelo_actual>Threshold_UserBottomVelo_PLC';
				moni_State:=-100;
		(*Left Î»ÖÃºÍËÙ¶È±È¶Ô*)
		ELSIF Diff_UserTBLeftPos_actual>Threshold_UserTBLeftPos_PLC  THEN
				Error:=TRUE;
				ErrorID:=605;
				ErrorDescription:='Diff_UserTBLeftPos_actual>Threshold_UserTBLeftPos_PLC';
				moni_State:=-100;
		ELSIF  Diff_UserTBLeftVelo_actual>Threshold_UserTBLeftVelo_PLC THEN
				Error:=TRUE;
				ErrorID:=606;
				ErrorDescription:='Diff_UserTBLeftVelo_actual>Threshold_UserTBLeftVelo_PLC';
				moni_State:=-100;
		(*Right Î»ÖÃºÍËÙ¶È±È¶Ô*)
		ELSIF Diff_UserTBRightPos_actual>Threshold_UserTBRightPos_PLC  THEN
				Error:=TRUE;
				ErrorID:=607;
				ErrorDescription:='Diff_UserTBRightPos_actual>Threshold_UserTBRightPos_PLC';
				moni_State:=-100;
		ELSIF  Diff_UserTBRightVelo_actual>Threshold_UserTBRightVelo_PLC THEN
				Error:=TRUE;
				ErrorID:=608;
				ErrorDescription:='Diff_UserTBRightVelo_actual>Threshold_UserTBRightVelo_PLC';
				moni_State:=-100;
		END_IF
		//
		IF Diff_UserInPos_actual >Threshold_UserInPos_PLC THEN
				Error:=TRUE;
				ErrorID:=609;
				ErrorDescription:='Diff_UserInPos_actual >Threshold_UserInPos_PLC';
				moni_State:=-100;
		ELSIF Diff_UserInVelo_actual>Threshold_UserInVelo_PLC  THEN
				Error:=TRUE;
				ErrorID:=610;
				ErrorDescription:='Diff_UserInVelo_actual>Threshold_UserInVelo_PLC';
				moni_State:=-100;
		(*Out Î»ÖÃºÍËÙ¶È±È¶Ô*)
		ELSIF Diff_UserOutPos_actual>Threshold_UserOutPos_PLC THEN
				Error:=TRUE;
				ErrorID:=611;
				ErrorDescription:='Diff_UserOutPos_actual>Threshold_UserOutPos_PLC';
				moni_State:=-100;
		ELSIF Diff_UserOutVelo_actual>Threshold_UserOutVelo_PLC  THEN
				Error:=TRUE;
				ErrorID:=612;
				ErrorDescription:='Diff_UserOutVelo_actual>Threshold_UserOutVelo_PLC';
				moni_State:=-100;
		(*Left Î»ÖÃºÍËÙ¶È±È¶Ô*)
		ELSIF Diff_UserIOLeftPos_actual>Threshold_UserIOLeftPos_PLC  THEN
				Error:=TRUE;
				ErrorID:=613;
				ErrorDescription:='Diff_UserIOLeftPos_actual>Threshold_UserIOLeftPos_PLC';
				moni_State:=-100;
		ELSIF  Diff_UserIOLeftVelo_actual>Threshold_UserIOLeftVelo_PLC THEN
				Error:=TRUE;
				ErrorID:=614;
				ErrorDescription:='Diff_UserIOLeftVelo_actual>Threshold_UserIOLeftVelo_PLC';
				moni_State:=-100;
		(*Right Î»ÖÃºÍËÙ¶È±È¶Ô*)
		ELSIF Diff_UserIORightPos_actual>Threshold_UserIORightPos_PLC  THEN
				Error:=TRUE;
				ErrorID:=615;
				ErrorDescription:='Diff_UserIORightPos_actual>Threshold_UserIORightPos_PLC';
				moni_State:=-100;
		ELSIF  Diff_UserIORightVelo_actual>Threshold_UserIORightVelo_PLC THEN
				Error:=TRUE;
				ErrorID:=616;
				ErrorDescription:='Diff_UserIORightVelo_actual>Threshold_UserIORightVelo_PLC';
				moni_State:=-100;
		END_IF
-100:
		btn_UserGapStop:=TRUE;
		FB_PlcEmergencyStop();
		Error:=TRUE;
		LED_Error:=TRUE;
END_CASE
END_IF
END_ACTION

ACTION A_OneKeyToMaxGap:
//0.上升沿触发
//1.判断电机是否在开启状态,没有就打开电源
//2.判断是否在Moving状态,若有就Stop
//3.将磁间隙打开到至最大阈值
//4.到位后给出反馈
OneKeyToMaxGap_RTRIG(CLK:=btn_OneKeyToMaxGap);
IF OneKeyToMaxGap_RTRIG.Q THEN
	OneKeyToMaxGap_Triggered:=TRUE;
	OneKeyToMaxGap_Done:=FALSE;
END_IF
IF OneKeyToMaxGap_Triggered THEN
	CASE OneKeyToMaxGap_State OF
		0://1.判断电机是否在开启状态,没有就打开电源
			IF st_Power=1 THEN
				OneKeyToMaxGap_State:=1;
			ELSE
				btn_PowerOn:=TRUE;
				IF btn_PowerOn THEN
					A_PowerOn();
				END_IF
			END_IF
		1://1.判断是否在谱学扫描模式，如果是，则切换回正常运动模式
			IF IsSSMotionMode THEN
				SS_Stop:=TRUE;
				IsSSMotionMode:=FALSE;
			END_IF
			OneKeyToMaxGap_State:=2;
		2://判断是否在taper，如果在taper,则判断是否在运动，如果是，则停止运动,0.5sh后，转入下一步
			IF TaperOrNot THEN
				IF moveStatusLeftTop OR moveStatusRightTop OR moveStatusLeftBottom OR moveStatusRightBottom THEN
					btn_UserGapStop:=TRUE;
				ELSE
					OneKeyToMaxGap_TON_Stop2Move_InTaperMode(PT:=T#0.5S);
					OneKeyToMaxGap_TON_Stop2Move_InTaperMode.IN:=TRUE;
					IF OneKeyToMaxGap_TON_Stop2Move_InTaperMode.Q THEN
						TaperOrNot:=FALSE;//关闭taper模式
						OneKeyToMaxGap_State:=3;
						OneKeyToMaxGap_TON_Stop2Move_InTaperMode.IN:=FALSE;
					END_IF
				END_IF
			ELSE
				OneKeyToMaxGap_State:=3;
			END_IF
		3://3.判断是否在Moving状态,若有就Stop.Taper模式已处理完，此处开始走正常GAP开合逻辑
			IF moveStatusLeftTop OR moveStatusRightTop OR moveStatusLeftBottom OR moveStatusRightBottom THEN
				btn_UserGapStop:=TRUE;
			ELSE
				OneKeyToMaxGap_TON_Stop2Move(PT:=T#0.5S);
				OneKeyToMaxGap_TON_Stop2Move.IN:=TRUE;
				IF OneKeyToMaxGap_TON_Stop2Move.Q THEN
					OneKeyToMaxGap_State:=4;
					OneKeyToMaxGap_TON_Stop2Move.IN:=FALSE;
				END_IF
			END_IF
		4://4.将磁间隙打开到至最大阈值
			OneKeyToMaxGap_TON(PT:=INT_TO_TIME(LREAL_TO_INT(max_UserGapPositionNew+30))*1000);
			OneKeyToMaxGap_TON.IN:=TRUE;
			OneKeyToMaxGap_TON_Power2Move(PT:=T#0.1S);
			OneKeyToMaxGap_TON_Power2Move.IN:=TRUE;
			UserGapPositionNew:=max_UserGapPositionNew;
			UserGapVelocityNew:=1;
			btn_UserGapMove:=TRUE;
			IF OneKeyToMaxGap_TON_Power2Move.Q THEN
				OneKeyToMaxGap_TON_Power2Move.IN:=FALSE;
				IF FB_MOVE.BCGapDone THEN
					OneKeyToMaxGap_State:=88;
				END_IF
			END_IF
			IF OneKeyToMaxGap_TON.Q THEN//如果150s后，还没有运动到指定gap，则报错
				OneKeyToMaxGap_TON.IN:=FALSE;
				OneKeyToMaxGap_State:=-100;
			END_IF
			IF  btn_UserGapStop THEN
				//
				OneKeyToMaxGap_State:=0;
				OneKeyToMaxGap_Triggered:=FALSE;
				btn_OneKeyToMaxGap:=FALSE;
				OneKeyToMaxGap_Triggered:=FALSE;
				OneKeyToMaxGap_State:=0;
			END_IF
		88://6.到位后给出反馈
			OneKeyToMaxGap_Done:=TRUE;	
			Error:=FALSE;
			ErrorID:=0;
			ErrorDescription:='';
			btn_OneKeyToMaxGap:=FALSE;
			OneKeyToMaxGap_Triggered:=FALSE;
			OneKeyToMaxGap_State:=0;
				
		-100:
			OneKeyToMaxGap_Done:=FALSE;
			Error:=TRUE;
			ErrorID:=1705;
			ErrorDescription:='OneKeyToMaxGap Fail';
			btn_OneKeyToMaxGap:=FALSE;
			OneKeyToMaxGap_Triggered:=FALSE;
			OneKeyToMaxGap_State:=0;
	END_CASE
END_IF
END_ACTION

ACTION A_PowerOff:
CASE d_state OF
		0:(*PowerOff*)
			FB_Power(Off:=TRUE);
				d_state:=1;
		1:
			IF NOT FB_power.OffStatus THEN
				d_state:=1;
			ELSE
				d_state:=88;
			END_IF
		88:(*ResetAllState*)
			btn_PowerOn:=FALSE;
			btn_UserGapMove:=FALSE;
			btn_UserGapStop:=FALSE;
			fb_ton1.IN:=FALSE;
			fb_ton2.IN:=FALSE;
			fb_ton3.IN:=FALSE;
			State:=0;
			Busy:=FALSE;
			InitPowerDone:=FALSE;
			InitCompensationDatasDone:=FALSE;
			Error:=FALSE;
			ErrorID:=0;
			m_state:=0;
			n_state:=0;
			s_state:=0;
			btn_PowerOff:=FALSE;
			d_state:=0;
			Led_Run:=FALSE;
			Led_Error:=FALSE;
			moni_State:=0;
			i:=0;
END_CASE
END_ACTION

ACTION A_PowerOn:
(****************************************************************
NAME:			A_PowerOn
DATA:			2018.1.9
VERSION:		1.0.0
DESCRIPTION:	
				ÉÏµãÃüÁîºó£¬Ë³ÐòÖ´ÐÐ£º
				1.FB_PowerOn
				·µ»ØÖ´ÐÐÊÇ·ñ³É¹¦
HISTORY:
				2019.1.9		NEW

***************************************************************)
fb_ton3(PT:=t#0.5s);
CASE State OF
	0:	(*FB_Power_On*)
		FB_Power(On:=TRUE);
		fb_ton3.IN:=TRUE;
		State:=1;
	1:	(*wait*)
		FB_power();
		IF NOT FB_power.OnStatus THEN		(*FB_Power_OnÃ»ÓÐÖ´ÐÐÍê£¬wait£¬³¬Ê±FB Error*)
			IF NOT fb_ton3.Q THEN
				State:=1;
			ELSE
				ErrorID:=1;
				State:=99;
			END_IF
		ELSE
			State:=88;
		END_IF
	88:	(*All Done*)
		btn_PowerOn:=FALSE;
		State:=0;
		Error:=FALSE;
		ErrorID:=0;
		Busy:=FALSE;
		InitPowerDone:=TRUE;
		FB_power.On:=FALSE;
		fb_ton3.IN:=FALSE;
		LED_Error:=FALSE;
	99:
		Error:=TRUE;
		//ErrorID:=701;
		//ErrorDescription:='power on error';		
		btn_PowerOn:=FALSE;
		State:=99;
		Busy:=FALSE;
		InitPowerDone:=FALSE;
		fb_ton3.IN:=FALSE;
		LED_Error:=TRUE;
END_CASE
END_ACTION

ACTION A_RegularMotion:
(*如果该ID没有taper需求，则TaperFunctionSolidOn=FALSE，则判定taperOrNot为false*)
IF NOT TaperFunctionSolidOn THEN
	TaperOrNot:=FALSE;
END_IF
(*若GAP将有变化，首先检测TAPER是否超出阈值，若超出，则报错，提示必须先将TAPER回归到0，才可以改变GAP*)
IF NOT (Global_ChainProtection_MPS_Triggered OR Global_ChainProtection_EPS_Triggered) THEN//在触发联锁保护后，taper保护关闭
	IF ABS(UserGapPositionNew-UserGapPositionDisplay)>Threshold_GapChangeFlag AND btn_UserGapMove THEN
		IF UserTaperPositionDisplay>Threshold_TaperChangeFlag THEN
			btn_UserGapStop:=TRUE;
			btn_UserGapMove:=FALSE;
			Error:=TRUE;
			ErrorId:=809;
			ErrorDescription:='Please Move Taper to zero first before move gap';
			RETURN;
		END_IF
	END_IF
END_IF
(*Taper和gap连锁限制性保护。比如11mm时候如果taper，入口端gap变小，会有压真空盒的问题。设置保护*)
IF NOT (Global_ChainProtection_MPS_Triggered OR Global_ChainProtection_EPS_Triggered)  THEN//在触发联锁保护后，taper保护关闭
	IF taperOrNot THEN 	
		IF UserGapPositionNew-TaperAndGapSafetyfactor*TaperAndGapSafetyScale*UserTaperPositionNew<=(min_UserGapPositionNew+TaperAndGapSafetyMinGapMargin)
		 AND btn_UserGapMove THEN
			btn_UserGapStop:=TRUE;
			btn_UserGapMove:=FALSE;
			Error:=TRUE;
			ErrorId:=810;
			ErrorDescription:='Target taper is too big at current Gap';
			RETURN;
		END_IF
	END_IF
END_IF
(*分别比较四轴目标位置与当前位置的差，如果目标位置比当前位置低，则需要运动到更低-回程差一半；再运动至最终目标位置*)
//只在m=和n=0的时候判断，否则会出现一些BUG，比如往大间隙开时，运动到位后m不能回到0.
IF m_state=0 AND n_state=0 THEN
		TargetPosLessThanCurrentPos:=FALSE;
	IF LeftTopLinPositionNew-Pos_LeftTopLin<-LEDriftErrorThreshold THEN
			TargetPosLessThanCurrentPos:=TRUE;
			TargetLTPosLessThanCurrentLTPos:=TRUE;
	ELSE
			TargetLTPosLessThanCurrentLTPos:=FALSE;
	END_IF
	IF RightTopLinPositionNew-Pos_RightTopLin<-LEDriftErrorThreshold THEN
			TargetPosLessThanCurrentPos:=TRUE;
			TargetRTPosLessThanCurrentRTPos:=TRUE;
	ELSE
			TargetRTPosLessThanCurrentRTPos:=FALSE;
	END_IF
	IF LeftBottomLinPositionNew-Pos_LeftBottomLin<-LEDriftErrorThreshold THEN
			TargetPosLessThanCurrentPos:=TRUE;
			TargetLBPosLessThanCurrentLBPos:=TRUE;
	ELSE
			TargetLBPosLessThanCurrentLBPos:=FALSE;
	END_IF
	IF RightBottomLinPositionNew-Pos_RightBottomLin<-LEDriftErrorThreshold THEN
			TargetPosLessThanCurrentPos:=TRUE;
			TargetRBPosLessThanCurrentRBPos:=TRUE;
	ELSE
			TargetRBPosLessThanCurrentRBPos:=FALSE;
	END_IF
	IF LeftInLinPositionNew-Pos_LeftInLin<-LEDriftErrorThreshold THEN
			TargetPosLessThanCurrentPos:=TRUE;
			TargetLIPosLessThanCurrentLIPos:=TRUE;
	ELSE
			TargetLIPosLessThanCurrentLIPos:=FALSE;
	END_IF
	IF RightInLinPositionNew-Pos_RightInLin<-LEDriftErrorThreshold THEN
			TargetPosLessThanCurrentPos:=TRUE;
			TargetRIPosLessThanCurrentRIPos:=TRUE;
	ELSE
			TargetRIPosLessThanCurrentRIPos:=FALSE;
	END_IF
	IF LeftOutLinPositionNew-Pos_LeftOutLin<-LEDriftErrorThreshold THEN
			TargetPosLessThanCurrentPos:=TRUE;
			TargetLOPosLessThanCurrentLOPos:=TRUE;
	ELSE
			TargetLOPosLessThanCurrentLOPos:=FALSE;
	END_IF
	IF RightOutLinPositionNew-Pos_RightOutLin<-LEDriftErrorThreshold THEN
			TargetPosLessThanCurrentPos:=TRUE;
			TargetROPosLessThanCurrentROPos:=TRUE;
	ELSE
			TargetROPosLessThanCurrentROPos:=FALSE;
	END_IF
END_IF

(*Move*)
IF InitCompensationDatasDone THEN
		(*四轴目标位置都大于当前位置，直接走到目标位置即可，不需要先走到考虑回城误差的临时位置*)
		IF NOT TargetPosLessThanCurrentPos AND NOT HysteresisMoving THEN
			CASE m_state OF
				0:
					FB_Move.Mode:=5;						//1.gap;2.single;3.taper;4.debug;5.BCGap&UserMode
					FB_Move.CoupleState:=st_Couple;			
					FB_Move.PowerState:=st_Power;						
			
					IF btn_UserGapMove THEN
						IF NOT st_Power THEN
							ErrorID:=1501;
							Error:=TRUE;
							ErrorDescription:='Plz PowerOn Frist';
							LED_Error:=TRUE;
							//btn_UserGapMove:=FALSE;
							RETURN;
						ELSE
							ErrorID:=0;
							Error:=FALSE;
							ErrorDescription:='';
							LED_Error:=FALSE;
							//btn_UserGapMove:=TRUE;
						END_IF
						//目标速度位置赋值
						FB_Move.BCLeftTopPosition:=LeftTopLinPositionNew;
						FB_Move.BCRightTopPosition:=RightTopLinPositionNew;
						FB_Move.BCLeftBottomPosition:=LeftBottomLinPositionNew;
						FB_Move.BCRightBottomPosition:=RightBottomLinPositionNew;
						FB_Move.BCLeftInPosition:=LeftInLinPositionNew;
						FB_Move.BCRightInPosition:=RightInLinPositionNew;
						FB_Move.BCLeftOutPosition:=LeftOutLinPositionNew;
						FB_Move.BCRightOutPosition:=RightOutLinPositionNew;
						IF NOT TaperOrNot THEN
							FB_Move.BCLeftTopVelocity:=UserGapVelocityNew/2;
							FB_Move.BCRightTopVelocity:=UserGapVelocityNew/2;
							FB_Move.BCLeftBottomVelocity:=UserGapVelocityNew/2;
							FB_Move.BCRightBottomVelocity:=UserGapVelocityNew/2;
							FB_Move.BCLeftInVelocity:=UserGapVelocityNew/2;
							FB_Move.BCRightInVelocity:=UserGapVelocityNew/2;
							FB_Move.BCLeftOutVelocity:=UserGapVelocityNew/2;
							FB_Move.BCRightOutVelocity:=UserGapVelocityNew/2;
						ELSE
							FB_Move.BCLeftTopVelocity:=UserTaperVelocityNew;
							FB_Move.BCRightTopVelocity:=UserTaperVelocityNew;
							FB_Move.BCLeftBottomVelocity:=UserTaperVelocityNew;
							FB_Move.BCRightBottomVelocity:=UserTaperVelocityNew;
							FB_Move.BCLeftInVelocity:=UserTaperVelocityNew;
							FB_Move.BCRightInVelocity:=UserTaperVelocityNew;
							FB_Move.BCLeftOutVelocity:=UserTaperVelocityNew;
							FB_Move.BCRightOutVelocity:=UserTaperVelocityNew;
						END_IF
							FB_Move.BCGapMove:=TRUE;
							m_state:=1;
							FB_Move();
					END_IF
				1:
					btn_UserGapMove:=FALSE;
					FB_Move();
					IF NOT FB_Move.BCGapDone THEN
						Led_Run:=TRUE;
						m_state:=1;
					ELSE
						m_state:=88;
					END_IF
				88:
					btn_UserGapMove:=FALSE;
					Led_Run:=FALSE;
					m_state:=0;
			END_CASE
		(*四轴有目标位置小于当前位置，先走到临时位置，再走到目标位置*)
		ELSE
			CASE n_state OF
				0:
					FB_Move.Mode:=5;						//1.gap;2.single;3.taper;4.debug;5.BCGap&UserMode;5:userMode_2
					FB_Move.CoupleState:=st_Couple;			
					FB_Move.PowerState:=st_Power;			
					IF btn_UserGapMove THEN	
						IF NOT st_Power THEN
							ErrorID:=1501;
							Error:=TRUE;
							ErrorDescription:='Plz PowerOn Frist';
							LED_Error:=TRUE;
							//btn_UserGapMove:=FALSE;
							RETURN;
						ELSE
							ErrorID:=0;
							Error:=FALSE;
							ErrorDescription:='';
							LED_Error:=FALSE;
							//btn_UserGapMove:=TRUE;
						END_IF						
						//
						IF TargetLTPosLessThanCurrentLTPos THEN			
							FB_Move.BCLeftTopPosition:=LeftTopLinPositionNew-HysteresisError/2;
						ELSE
							FB_Move.BCLeftTopPosition:=LeftTopLinPositionNew;	
						END_IF
						//
						IF TargetRTPosLessThanCurrentRTPos THEN 
							FB_Move.BCRightTopPosition:=RightTopLinPositionNew-HysteresisError/2;
						ELSE					
							FB_Move.BCRightTopPosition:=RightTopLinPositionNew;
						END_IF
						//
						IF TargetLBPosLessThanCurrentLBPos THEN
							FB_Move.BCLeftBottomPosition:=LeftBottomLinPositionNew-HysteresisError/2;
						ELSE
							FB_Move.BCLeftBottomPosition:=LeftBottomLinPositionNew;
						END_IF
						//
						IF TargetRBPosLessThanCurrentRBPos THEN
							FB_Move.BCRightBottomPosition:=RightBottomLinPositionNew-HysteresisError/2;
						ELSE
							FB_Move.BCRightBottomPosition:=RightBottomLinPositionNew;
						END_IF						
						//
						IF TargetLIPosLessThanCurrentLIPos THEN			
							FB_Move.BCLeftInPosition:=LeftInLinPositionNew-HysteresisError/2;
						ELSE
							FB_Move.BCLeftInPosition:=LeftInLinPositionNew;	
						END_IF
						//
						IF TargetRIPosLessThanCurrentRIPos THEN 
							FB_Move.BCRightInPosition:=RightInLinPositionNew-HysteresisError/2;
						ELSE					
							FB_Move.BCRightInPosition:=RightInLinPositionNew;
						END_IF
						//
						IF TargetLOPosLessThanCurrentLOPos THEN
							FB_Move.BCLeftOutPosition:=LeftOutLinPositionNew-HysteresisError/2;
						ELSE
							FB_Move.BCLeftOutPosition:=LeftOutLinPositionNew;
						END_IF
						//
						IF TargetROPosLessThanCurrentROPos THEN
							FB_Move.BCRightOutPosition:=RightOutLinPositionNew-HysteresisError/2;
						ELSE
							FB_Move.BCRightOutPosition:=RightOutLinPositionNew;
						END_IF		
						//	close gap情况下，加入了LeftTopLinPositionNewTemp。//
						//如果在往小间隙运行过程中，改变了目标gap，会在第到达第一次目标位置后，继续向第二
						//次输入的目标运动，而不会回到第一次的目标位置。用temp锁定目标位置
						LeftTopLinPositionNewTemp:=LeftTopLinPositionNew;
						RightTopLinPositionNewTemp:=RightTopLinPositionNew;
						LeftBottomLinPositionNewTemp:=LeftBottomLinPositionNew;
						RightBottomLinPositionNewTemp:=RightBottomLinPositionNew;
						LeftInLinPositionNewTemp:=LeftInLinPositionNew;
						RightInLinPositionNewTemp:=RightInLinPositionNew;
						LeftOutLinPositionNewTemp:=LeftOutLinPositionNew;
						RightOutLinPositionNewTemp:=RightOutLinPositionNew;
			
						//
						IF NOT TaperOrNot THEN
							FB_Move.BCLeftTopVelocity:=UserGapVelocityNew/2;
							FB_Move.BCRightTopVelocity:=UserGapVelocityNew/2;
							FB_Move.BCLeftBottomVelocity:=UserGapVelocityNew/2;
							FB_Move.BCRightBottomVelocity:=UserGapVelocityNew/2;
							FB_Move.BCLeftInVelocity:=UserGapVelocityNew/2;
							FB_Move.BCRightInVelocity:=UserGapVelocityNew/2;
							FB_Move.BCLeftOutVelocity:=UserGapVelocityNew/2;
							FB_Move.BCRightOutVelocity:=UserGapVelocityNew/2;
							IF UserGapVelocityNew >1 THEN								  
								ErrorID:=1502;
								Error:=TRUE;
								ErrorDescription:='UserGapVelocityNew must<=1';
								LED_Error:=TRUE;
								btn_UserGapMove:=FALSE;
								RETURN;
							ELSE
								ErrorID:=0;
								Error:=FALSE;
								ErrorDescription:='';
								LED_Error:=FALSE;	
							END_IF									
						ELSE
							FB_Move.BCLeftTopVelocity:=UserTaperVelocityNew;
							FB_Move.BCRightTopVelocity:=UserTaperVelocityNew;
							FB_Move.BCLeftBottomVelocity:=UserTaperVelocityNew;
							FB_Move.BCRightBottomVelocity:=UserTaperVelocityNew;
							FB_Move.BCLeftInVelocity:=UserTaperVelocityNew;
							FB_Move.BCRightInVelocity:=UserTaperVelocityNew;
							FB_Move.BCLeftOutVelocity:=UserTaperVelocityNew;
							FB_Move.BCRightOutVelocity:=UserTaperVelocityNew;
						END_IF	

						FB_Move.BCGapMove:=TRUE;
						FB_Move();
						HysteresisMoving:=TRUE;		
						n_state:=1;	
					END_IF
				1:
					btn_UserGapMove:=FALSE;
					FB_Move();
					IF NOT FB_Move.BCGapDone THEN			(*还未运动到位置,运动过程中*)
						Led_Run:=TRUE;
						n_state:=1;
					ELSE									
						n_state:=2;							(*转到下一步，运动到最终位置*)
						FB_Move.BCGapMove:=FALSE;
						//Led_Run:=FALSE;
					END_IF
				2:
					FB_Move.BCGapReset:=FALSE;
					FB_Move.Mode:=5;						//1.gap;2.single;3.taper;4.debug;5.BCGap&UserMode
					FB_Move.CoupleState:=st_Couple;			
					FB_Move.PowerState:=st_Power;			
					FB_Move.BCGapMove:=TRUE;
					//直接走到目标位置，已经走到位置的，可以继续下命令，只不过它不在走了而已
					FB_Move.BCLeftTopPosition:=LeftTopLinPositionNewTemp;	
					FB_Move.BCRightTopPosition:=RightTopLinPositionNewTemp;
					FB_Move.BCLeftBottomPosition:=LeftBottomLinPositionNewTemp;
					FB_Move.BCRightBottomPosition:=RightBottomLinPositionNewTemp;
					FB_Move.BCLeftInPosition:=LeftInLinPositionNewTemp;	
					FB_Move.BCRightInPosition:=RightInLinPositionNewTemp;
					FB_Move.BCLeftOutPosition:=LeftOutLinPositionNewTemp;
					FB_Move.BCRightOutPosition:=RightOutLinPositionNewTemp;
					//
					IF NOT TaperOrNot THEN
						FB_Move.BCLeftTopVelocity:=UserGapVelocityNew/2;
						FB_Move.BCRightTopVelocity:=UserGapVelocityNew/2;
						FB_Move.BCLeftBottomVelocity:=UserGapVelocityNew/2;
						FB_Move.BCRightBottomVelocity:=UserGapVelocityNew/2;
						FB_Move.BCLeftInVelocity:=UserGapVelocityNew/2;
						FB_Move.BCRightInVelocity:=UserGapVelocityNew/2;
						FB_Move.BCLeftOutVelocity:=UserGapVelocityNew/2;
						FB_Move.BCRightOutVelocity:=UserGapVelocityNew/2;
					ELSE
						FB_Move.BCLeftTopVelocity:=UserTaperVelocityNew;
						FB_Move.BCRightTopVelocity:=UserTaperVelocityNew;
						FB_Move.BCLeftBottomVelocity:=UserTaperVelocityNew;
						FB_Move.BCRightBottomVelocity:=UserTaperVelocityNew;
						FB_Move.BCLeftInVelocity:=UserTaperVelocityNew;
						FB_Move.BCRightInVelocity:=UserTaperVelocityNew;
						FB_Move.BCLeftOutVelocity:=UserTaperVelocityNew;
						FB_Move.BCRightOutVelocity:=UserTaperVelocityNew;
					END_IF
					FB_Move();							
					n_state:=3;
				3:
					FB_Move();
					IF NOT FB_Move.BCGapDone THEN			(*还未运动到位置,运动过程中*)
						Led_Run:=TRUE;
						n_state:=3;
					ELSE									
						n_state:=88;							(*运动到了最终位置*)
					END_IF
					(*
					IF NOT Unreach_LS_Bottom THEN
						n_state:=88;							(*在运动过程中如果碰到下限位，则也转到下一步，运动到最终位置*)
						FB_Move.BCGapMove_2:=FALSE;
					END_IF
					*)
				88:
					btn_UserGapMove:=FALSE;					
					Led_Run:=FALSE;
					n_state:=0;
					HysteresisMoving:=FALSE;
			END_CASE
		END_IF
	//
	//FB_Move.BCLeftTopPosition等四轴位置监控
	//
END_IF

IF btn_UserGapStop OR btn_Reset THEN
	FB_Move.BCGapReset:=TRUE;
	FB_Move();	
	btn_UserGapMove:=FALSE;	
	m_state:=0;	
	n_state:=0;	
	HysteresisMoving:=FALSE;
	CASE s_state OF
			0:
				FB_Stop.Mode:=5;	
				FB_Stop.CoupleState:=st_Couple;	
				FB_Stop.PowerState:=st_Power;
				FB_Stop.BCGapStop:=TRUE;
				FB_Stop();	
				s_state:=1;
			1:
				FB_Stop();
				IF NOT FB_Stop.BCGapDone THEN
					s_state:=1;
				ELSE
					s_state:=88;
				END_IF
			88:
				btn_UserGapStop:=FALSE;	
				FB_Move.BCGapReset:=FALSE;
				btn_reset:=FALSE;
				s_state:=0;
		END_CASE
END_IF

(*触发限位开关后，相当于点击了Stop按钮*)
FTrig_ReachLS(CLK:=Unreach_LS_Far AND Unreach_LS_Near);
IF FTrig_ReachLS.Q THEN
	btn_UserGapStop:=TRUE;
END_IF
END_ACTION

ACTION A_SpectroscopyScanningMotion:
(*
(*输入保护*)
IF SS_Move AND SSMotionMode AND NOT RegularMotionMode THEN
	IF NOT inRange_SS_StepSize THEN
		SS_Stop:=TRUE;
		SS_Move:=FALSE;
		Error:=TRUE;
		ErrorId:=805;
		ErrorDescription:='target StepSize out of range,please check';
		RETURN;
	ELSE
		SS_Stop:=FALSE;
		Error:=FALSE;
		ErrorId:=0;
		ErrorDescription:='';	
	END_IF
	//
	IF NOT inRange_SS_StepNumber THEN
		SS_Stop:=TRUE;
		SS_Move:=FALSE;
		Error:=TRUE;
		ErrorId:=806;
		ErrorDescription:='target StepNumber out of range,please check';
		RETURN;
	ELSE
		SS_Stop:=FALSE;
		Error:=FALSE;
		ErrorId:=0;
		ErrorDescription:='';	
	END_IF
	IF NOT inRange_SS_StepVelocity THEN
		SS_Stop:=TRUE;
		SS_Move:=FALSE;
		Error:=TRUE;
		ErrorId:=807;
		ErrorDescription:='target StepVelocity out of range,please check';
		RETURN;
	ELSE
		SS_Stop:=FALSE;
		Error:=FALSE;
		ErrorId:=0;
		ErrorDescription:='';	
	END_IF
	IF NOT inRange_StepEachTime_ms THEN
		SS_Stop:=TRUE;
		SS_Move:=FALSE;
		Error:=TRUE;
		ErrorId:=808;
		ErrorDescription:='target StepEachTime_ms out of range,please check';
		RETURN;
	ELSE
		SS_Stop:=FALSE;
		Error:=FALSE;
		ErrorId:=0;
		ErrorDescription:='';	
	END_IF
END_IF
(*单步时长转换*)
StepEachTime:=INT_TO_TIME(StepEachTime_ms);
SS_TON(PT:=StepEachTime);
(*上升沿触发，初始SS位置=当前磁间隙*)
RTRG_SS_StartPositionDisplay(CLK:=SS_Move);
IF RTRG_SS_StartPositionDisplay.Q THEN
	SS_StartPositionDisplay:=UserGapPositionDisplay;
	SS_InitStartPositionDone:=TRUE;
END_IF
(*SS主程序*)
IF InitPowerDone AND InitCompensationDatasDone AND SS_Move AND SS_InitStartPositionDone THEN
	CASE SS_MoveState OF
		0:
				//UserGapPositionNew:=UserGapPositionDisplay+SS_StepSize;
				UserGapPositionNew:=SS_StartPositionDisplay+SS_StepSize*(SS_currentStep+1);
				A_InitCompensationData();
				FB_Move.Mode:=5;						//1.gap;2.single;3.taper;4.debug;5.BCGap&UserMode
				FB_Move.CoupleState:=st_Couple;			
				FB_Move.PowerState:=st_Power;							
				FB_Move.BCLeftTopPosition:=LeftTopLinPositionNew;
				FB_Move.BCLeftTopVelocity:=UserGapVelocityNew/2;
				FB_Move.BCRightTopPosition:=RightTopLinPositionNew;
				FB_Move.BCRightTopVelocity:=UserGapVelocityNew/2;
				FB_Move.BCLeftBottomPosition:=LeftBottomLinPositionNew;
				FB_Move.BCLeftBottomVelocity:=UserGapVelocityNew/2;
				FB_Move.BCRightBottomPosition:=RightBottomLinPositionNew;
				FB_Move.BCRightBottomVelocity:=UserGapVelocityNew/2;		
				FB_Move.BCGapMove:=TRUE;
				FB_Move();
				SS_MoveState:=1;
		1:
				SS_TON.IN:=TRUE;
				FB_Move();
				IF FB_Move.GapMoving AND NOT SS_TimeCountBegin THEN
					SS_StepSystemTime_Begin[SS_currentStep]:=F_GetSysTime();
					SS_TimeCountBegin:=TRUE;
				END_IF
				IF NOT FB_Move.BCGapDone THEN			
					Led_Run:=TRUE;
					SS_MoveState:=1;
				ELSE									
					SS_MoveState:=66;
					SS_StepSystemTime_End[SS_currentStep]:=F_GetSysTime();
					SS_StepCountTime[SS_currentStep]:=SS_StepSystemTime_End[SS_currentStep]-SS_StepSystemTime_Begin[SS_currentStep];
					SS_TimeCountBegin:=FALSE;
				END_IF
		66:
				SS_currentStep:=SS_currentStep+1;			
				Led_Run:=FALSE;
				IF SS_currentStep=SS_StepNumber THEN								
					SS_MoveState:=88;
				END_IF
				IF SS_currentStep<SS_StepNumber THEN
					SS_MoveState:=77;
				END_IF
		77://等待单步时长够
				IF SS_TON.Q THEN
					SS_TON.IN:=FALSE;
					SS_MoveState:=0;
				END_IF
		88:
				SS_TON.IN:=FALSE;
				SS_Move:=FALSE;	
				Led_Run:=FALSE;
				SS_MoveState:=0;
				SS_currentStep:=0;
				SS_InitStartPositionDone:=FALSE;
				//SS_StepSystemTime[SS_StepNumber]:=F_GetSysTime();
	END_CASE
END_IF
(*获取每一步耗时*)
//FOR	m:= 0 TO SS_StepNumber DO
//	SS_StepCountTime[m]:=(SS_StepSystemTime_End[m]-SS_StepSystemTime_Begin[m]);
//END_FOR

(*STOP*)
IF SS_Stop THEN
	FB_Move.BCGapReset:=TRUE;							(*¸øÔË¶¯FB¸øÍ£Ö¹ÐÅºÅ£¬Ê¹FB_Move×´Ì¬»Ö¸´*)
	FB_Move();											(*Æô¶¯FB_Move*)
	SS_Move:=FALSE;								(*btn_GapMove:=FALSE*)
	SS_MoveState:=0;										(*m_state:=0;*)
	CASE SS_StopState OF
			0:
				FB_Stop.Mode:=5;							(*1£ºgapÄ£Ê½£»2£ºµ¥ÁºÄ£Ê½£»3£ºtaperÄ£Ê½£»4£ºDebugÄ£Ê½£»5£ºBCGapÄ£Ê½*)
				FB_Stop.CoupleState:=st_Couple;			(*ñîºÏ×´Ì¬ÊäÈë*)
				FB_Stop.PowerState:=st_Power;				(*µçÔ´×´Ì¬ÊäÈë*)
				FB_Stop.BCGapStop:=TRUE;				(*Execute TRUE*)
				FB_Stop();								(*Æô¶¯FB*)
				SS_StopState:=1;
			1:
				FB_Stop();
				IF NOT FB_Stop.BCGapDone THEN			(*Í£Ö¹Î´Íê³É£¬Ñ­»·*)
					SS_StopState:=1;
				ELSE									(*Í£Ö¹Íê³É£¬ÏÂÒ»²½*)
					SS_StopState:=88;
				END_IF
			88:
				SS_Stop:=FALSE;						(*»Ö¸´×´Ì¬*)
				FB_Move.BCGapReset:=FALSE;				(*ÔËÐÐFB*)
				SS_StopState:=0;
		END_CASE
END_IF

(*触发限位开关后，相当于点击了Stop按钮*)
FTrig_ReachLS(CLK:=Unreach_LS_Far AND Unreach_LS_Near);
IF FTrig_ReachLS.Q THEN
	SS_Stop:=TRUE;
END_IF
*)
END_ACTION

END_PROGRAM

// ---- POUs/CommonFB/MainFB/FB_Move.TcPOU
(****************************************************************
NAME:			FB_Move
DATA:			2017.2.17
VERSION:		1.0.0
DESCRIPTION:	FB_Move
HISTORY:
				2017.2.17		NEW
				2018.1.9		ÐÂÔöBCGapMode
***************************************************************)
FUNCTION_BLOCK FB_Move
VAR_INPUT
	(*È«¾Ö*)
	Mode:DINT;
	PowerState:BOOL;
	CoupleState:DINT;
	(*BCGapMode*)
	BCLeftTopPosition:LREAL;
	BCLeftTopVelocity:LREAL;
	BCRightTopPosition:LREAL;
	BCRightTopVelocity:LREAL;
	BCLeftBottomPosition:LREAL;
	BCLeftBottomVelocity:LREAL;
	BCRightBottomPosition:LREAL;
	BCRightBottomVelocity:LREAL;
	BCLeftInPosition:LREAL;
	BCLeftInVelocity:LREAL;
	BCRightInPosition:LREAL;
	BCRightInVelocity:LREAL;
	BCLeftOutPosition:LREAL;
	BCLeftOutVelocity:LREAL;
	BCRightOutPosition:LREAL;
	BCRightOutVelocity:LREAL;
	BCGapMove:BOOL;
	BCGapReset:BOOL;
	BCGapMove_2:BOOL;
	BCGapReset_2:BOOL;
	(*SingleCarrierMode*)
	TopPosition:LREAL;
	TopVelocity:LREAL;
	TopMove:BOOL;
	TopReset:BOOL;
	BottomPosition:LREAL;
	BottomVelocity:LREAL;
	BottomMove:BOOL;
	BottomReset:BOOL;
	InPosition:LREAL;
	InVelocity:LREAL;
	InMove:BOOL;
	InReset:BOOL;
	OutPosition:LREAL;
	OutVelocity:LREAL;
	OutMove:BOOL;
	OutReset:BOOL;
	(**DebugMode*)
	LeftTopPosition:LREAL;
	LeftTopVelocity:LREAL;
	LeftTopMove:BOOL;
	LeftTopStop:BOOL;
	LeftTopReset:BOOL;
	RightTopPosition:LREAL;
	RightTopVelocity:LREAL;
	RightTopMove:BOOL;
	RightTopStop:BOOL;
	RightTopReset:BOOL;
	LeftBottomPosition:LREAL;
	LeftBottomVelocity:LREAL;
	LeftBottomMove:BOOL;
	LeftBottomStop:BOOL;
	LeftBottomReset:BOOL;
	RightBottomPosition:LREAL;
	RightBottomVelocity:LREAL;
	RightBottomMove:BOOL;
	RightBottomStop:BOOL;
	RightBottomReset:BOOL;
	
	LeftInPosition:LREAL;
	LeftInVelocity:LREAL;
	LeftInMove:BOOL;
	LeftInStop:BOOL;
	LeftInReset:BOOL;
	RightInPosition:LREAL;
	RightInVelocity:LREAL;
	RightInMove:BOOL;
	RightInStop:BOOL;
	RightInReset:BOOL;
	LeftOutPosition:LREAL;
	LeftOutVelocity:LREAL;
	LeftOutMove:BOOL;
	LeftOutStop:BOOL;
	LeftOutReset:BOOL;
	RightOutPosition:LREAL;
	RightOutVelocity:LREAL;
	RightOutMove:BOOL;
	RightOutStop:BOOL;
	RightOutReset:BOOL;
END_VAR
VAR_OUTPUT
	FbID:DINT:=1001;
	GapState:DINT;
	GapBusy:BOOL;
	GapDone:BOOL;
	GapMoving:BOOL;

	BCGapState:DINT;
	BCGapBusy:BOOL;
	BCGapDone:BOOL;

	TopState:DINT;
	TopBusy:BOOL;
	TopDone:BOOL;
	BottomState:DINT;
	BottomBusy:BOOL;
	BottomDone:BOOL;
	
	InState:DINT;
	InBusy:BOOL;
	InDone:BOOL;
	OutState:DINT;
	OutBusy:BOOL;
	OutDone:BOOL;

	LeftTopState:DINT;
	LeftTopBusy:BOOL;
	LeftTopDone:BOOL;
	RightTopState:DINT;
	RightTopBusy:BOOL;
	RightTopDone:BOOL;
	LeftBottomState:DINT;
	LeftBottomBusy:BOOL;
	LeftBottomDone:BOOL;
	RightBottomState:DINT;
	RightBottomBusy:BOOL;
	RightBottomDone:BOOL;

	LeftInState:DINT;
	LeftInBusy:BOOL;
	LeftInDone:BOOL;
	RightInState:DINT;
	RightInBusy:BOOL;
	RightInDone:BOOL;
	LeftOutState:DINT;
	LeftOutBusy:BOOL;
	LeftOutDone:BOOL;
	RightOutState:DINT;
	RightOutBusy:BOOL;
	RightOutDone:BOOL;


	Error:BOOL;
	ErrorID:DINT;
	
	GapState_2:DINT;
	GapBusy_2:BOOL;
	GapDone_2:BOOL;

	BCGapState_2:DINT;
	BCGapBusy_2:BOOL;
	BCGapDone_2:BOOL;
END_VAR
VAR
	LeftTop_MC_MoveAbsolute: MC_MoveAbsolute;
	LeftBottom_MC_MoveAbsolute: MC_MoveAbsolute;
	RightTopLin_MC_MoveAbsolute: MC_MoveAbsolute;
	RightBottomLin_MC_MoveAbsolute: MC_MoveAbsolute;
	LeftIn_MC_MoveAbsolute: MC_MoveAbsolute;
	LeftOut_MC_MoveAbsolute: MC_MoveAbsolute;
	RightInLin_MC_MoveAbsolute: MC_MoveAbsolute;
	RightOutLin_MC_MoveAbsolute: MC_MoveAbsolute;
	fb_ton: TON;
	fb_ton1: TON;
	fb_ton2: TON;
	
	fb_ton3: TON;
	fb_ton4: TON;
	fb_ton_debug_1:TON;
	fb_ton_debug_2:TON;
	fb_ton_debug_3:TON;
	fb_ton_debug_4:TON;
	fb_ton_debug_5:TON;
	fb_ton_debug_6:TON;
	fb_ton_debug_7:TON;
	fb_ton_debug_8:TON;
	fb_ton_BC:TON;
	fb_ton_BC_2:TON;
END_VAR

IF PowerState=1 THEN
	IF Mode=1 AND TopMove THEN//Mode:=1,single carrier mode
		A_TopMove();
	ELSIF Mode=1 AND BottomMove THEN
		A_BottomMove();
	ELSIF Mode=1 AND InMove THEN
		A_InMove();
	ELSIF Mode=1 AND OutMove THEN
		A_OutMove();
	ELSIF Mode=2 AND LeftTopMove THEN//Mode:=2,Debug mode
		A_LeftTopMove();
	ELSIF Mode=2 AND RightTopMove THEN
		A_RightTopMove();
	ELSIF Mode=2 AND LeftBottomMove THEN
		A_LeftBottomMove();
	ELSIF Mode=2 AND RightBottomMove THEN
		A_RightBottomMove();
	ELSIF Mode=2 AND LeftInMove THEN
		A_LeftInMove();
	ELSIF Mode=2 AND RightInMove THEN
		A_RightInMove();
	ELSIF Mode=2 AND LeftOutMove THEN
		A_LeftOutMove();
	ELSIF Mode=2 AND RightOutMove THEN
		A_RightOutMove();
	ELSIF Mode=5 AND BCGapMove THEN//Mode:=5,userMode
		A_BCGapMove();
	END_IF
END_IF

ACTION A_BCGapMove:
IF BCGapMove THEN
BCGapBusy:=TRUE;
BCGapDone:=FALSE;
fb_ton_BC(PT:=t#80s);(*2mm/s max spees,120mmÐÐ³Ì£¬60sÄÚ×ßÍê*)

A_MoveMC();
IF  LeftTopLin.Status.Moving AND RightTopLin.Status.Moving
	AND LeftBottomLin.Status.Moving AND RightBottomLin.Status.Moving
	AND LeftInLin.Status.Moving AND RightInLin.Status.Moving
	AND LeftOutLin.Status.Moving AND RightOutLin.Status.Moving THEN
	GapMoving:=TRUE;
ELSE
	GapMoving:=FALSE;
END_IF
CASE BCGapState OF
	0:
		IF LeftTopLin.Status.Moving OR RightTopLin.Status.Moving
			OR LeftBottomLin.Status.Moving OR RightBottomLin.Status.Moving
			OR LeftInLin.Status.Moving OR RightInLin.Status.Moving
			OR LeftOutLin.Status.Moving OR RightOutLin.Status.Moving THEN	(*ÖáÕýÔÚÔËÐÐ£¬Ñ­»·¸Ã²½µÈ´ý*)
				BCGapState:=88;
		ELSIF LeftTop_MC_MoveAbsolute.Error OR LeftBottom_MC_MoveAbsolute.Error
			OR RightTopLin_MC_MoveAbsolute.Error OR RightBottomLin_MC_MoveAbsolute.Error
			OR LeftIn_MC_MoveAbsolute.Error OR LeftOut_MC_MoveAbsolute.Error
			OR RightInLin_MC_MoveAbsolute.Error OR RightOutLin_MC_MoveAbsolute.Error THEN	(*¼ì²éMC Error*)
				ErrorID:=2;
				BCGapState:=99;
		(*ELSIF ABS(Pos_LeftTopLin-GapPosition/2)<0.002 AND  ABS(Pos_LeftBottomLin-GapPosition)<0.002 THEN	(*Ä¿±êÎ»ÖÃÓëµ±Ç°Î»ÖÃÒ»Ñù£¬²»¶¯*)
			GapState:=88;*)
		ELSIF leftTopLin.Status.NotMoving AND  leftBottomLin.Status.NotMoving
			 AND RightTopLin.Status.NotMoving AND RightBottomLin.Status.NotMoving
			 AND leftInLin.Status.NotMoving AND  leftOutLin.Status.NotMoving
			 AND RightInLin.Status.NotMoving AND RightOutLin.Status.NotMoving THEN	(*Öá¶¼´¦ÓÚÍ£Ö¹×´Ì¬Ê±£¬×ªÏÂÒ»²½*)
			BCGapState:=1;
		END_IF
	1:
		LeftTop_MC_MoveAbsolute.Position:=BCLeftTopPosition;
		LeftTop_MC_MoveAbsolute.Velocity:=BCLeftTopVelocity;
		LeftBottom_MC_MoveAbsolute.Position:=BCLeftBottomPosition;
		LeftBottom_MC_MoveAbsolute.Velocity:=BCLeftBottomVelocity;
		RightTopLin_MC_MoveAbsolute.Position:=BCRightTopPosition;
		RightTopLin_MC_MoveAbsolute.Velocity:=BCRightTopVelocity;
		RightBottomLin_MC_MoveAbsolute.Position:=BCRightBottomPosition;
		RightBottomLin_MC_MoveAbsolute.Velocity:=BCRightBottomVelocity;
		LeftIn_MC_MoveAbsolute.Position:=BCLeftInPosition;
		LeftIn_MC_MoveAbsolute.Velocity:=BCLeftInVelocity;
		LeftOut_MC_MoveAbsolute.Position:=BCLeftOutPosition;
		LeftOut_MC_MoveAbsolute.Velocity:=BCLeftOutVelocity;
		RightInLin_MC_MoveAbsolute.Position:=BCRightInPosition;
		RightInLin_MC_MoveAbsolute.Velocity:=BCRightInVelocity;
		RightOutLin_MC_MoveAbsolute.Position:=BCRightOutPosition;
		RightOutLin_MC_MoveAbsolute.Velocity:=BCRightOutVelocity;
		LeftTop_MC_MoveAbsolute.Execute:=TRUE;
		LeftBottom_MC_MoveAbsolute.Execute:=TRUE;
		RightTopLin_MC_MoveAbsolute.Execute:=TRUE;
		RightBottomLin_MC_MoveAbsolute.Execute:=TRUE;
		LeftIn_MC_MoveAbsolute.Execute:=TRUE;
		LeftOut_MC_MoveAbsolute.Execute:=TRUE;
		RightInLin_MC_MoveAbsolute.Execute:=TRUE;
		RightOutLin_MC_MoveAbsolute.Execute:=TRUE;
		fb_ton_BC.IN:=TRUE;
		BCGapState:=2;
	2:
		IF NOT LeftTop_MC_MoveAbsolute.Done OR NOT  LeftBottom_MC_MoveAbsolute.Done
				OR NOT RightTopLin_MC_MoveAbsolute.Done OR NOT RightBottomLin_MC_MoveAbsolute.Done
				OR NOT LeftIn_MC_MoveAbsolute.Done OR NOT  LeftOut_MC_MoveAbsolute.Done
				OR NOT RightInLin_MC_MoveAbsolute.Done OR NOT RightOutLin_MC_MoveAbsolute.Done THEN		(*ÔË¶¯ÖÐ£¬¼ì²éDoneÐÅºÅ£¬Ã»ÓÐÔòÑ­»·*)
			BCGapState:=2;
		ELSIF LeftTop_MC_MoveAbsolute.Done  AND  LeftBottom_MC_MoveAbsolute.Done 
			AND RightTopLin_MC_MoveAbsolute.Done AND RightBottomLin_MC_MoveAbsolute.Done
			AND LeftIn_MC_MoveAbsolute.Done  AND  LeftOut_MC_MoveAbsolute.Done 
			AND RightInLin_MC_MoveAbsolute.Done AND RightOutLin_MC_MoveAbsolute.Done THEN		(*ÔË¶¯Íê³É£¬×ªÏÂÒ»²½*)
			BCGapState:=88;
		END_IF
		(*½ÓÊÕµ½stopÐÅºÅÊ±£¬reset×´Ì¬*)
		IF BCGapReset THEN
			BCGapState:=89;
		END_IF

